KUKA KRL program: Glode_HanGao.src, Glode_HanGao.dat

--- Glode_HanGao.src ---
&ACCESS RVO1
&REL 298
&PARAM EDITMASK = *
&PARAM TEMPLATE = C:\KRC\Roboter\Template\vorgabe
&PARAM DISKPATH = KRC:\R1\Program\HK
DEF Glode_HanGao( )

;# DATE:2021-1-4



END

GLOBAL DEF HanGao_Surr_Calculate(Surr_Path:IN , Sink_Area:IN ,POS_Type:IN , Lin_Pos:OUt , Cir_Middle_POS:OUT , Cir_END_POS:OUT , Offset_info:OUT  ,Offset_cir_info:out , Offset_No:IN , Work_Area:IN, Sink_Type:IN)
;------------DECL_VALUE--------------
DECL REAL Surr_Path
DECL Sink_Type_Enum  Sink_Type
DECL Area_Enum Sink_Area
DECL E6POS Lin_Pos
DECL E6POS Cir_Middle_POS
DECL E6POS Cir_END_POS
DECL Pos_Type_Enum Pos_Type
DECL Offset_POS Offset_info , Offset_cir_info
DECL Surround_Welding_Type Sink_Welding_Size
DECL INT OFFSET_NO,Work_Area

;------------DECL_VALUE--------------





Lin_Pos={X 0,Y 0, Z 0,A 0,B 0,C 0}

Cir_Middle_POS={X 0,Y 0, Z 0,A 0,B 0,C 0}

Cir_END_POS={X 0,Y 0, Z 0,A 0,B 0,C 0}


switch Work_Area

CASE 1
Sink_Welding_Size=N1_Sink_Data

CASE 2
Sink_Welding_Size=N2_Sink_Data

ENDSWITCH



SWITCH Sink_Area

CASE #L0





 UL_Equation(N315_OFFSET_POS,N45_OFFSET_POS,(Surr_Path*0.01),Sink_Welding_Size.Sink_Size_R,Lin_Pos)



 ;Lin_Pos.X=Sink_Welding_Size.Sink_Size_Width+Sink_Welding_Size.Sink_Size_Down_Distance
 ;Lin_Pos.Y=(Sink_Welding_Size.Sink_Size_Long-Sink_Welding_Size.Sink_Size_R*2)* (1-(Surr_Path*0.01))+Sink_Welding_Size.Sink_Size_Left_Distance+Sink_Welding_Size.Sink_Size_R
 Lin_Pos.Z=-(Sink_Welding_Size.Sink_Size_Panel_Thick)

 Lin_Pos.A=0
 Lin_Pos.B=L0_Welding_Craft[Work_Area,OFFSET_NO].Welding_Angle
 Lin_Pos.C=0


L0_Welding_Craft[Work_Area,OFFSET_NO].Welding_Pos.X=Lin_Pos.X
L0_Welding_Craft[Work_Area,OFFSET_NO].Welding_Pos.Y=Lin_Pos.Y
L0_Welding_Craft[Work_Area,OFFSET_NO].Welding_Pos.Z=Lin_Pos.Z
L0_Welding_Craft[Work_Area,OFFSET_NO].Welding_Pos.A=Lin_Pos.A
L0_Welding_Craft[Work_Area,OFFSET_NO].Welding_Pos.B=Lin_Pos.B
L0_Welding_Craft[Work_Area,OFFSET_NO].Welding_Pos.C=Lin_Pos.C
CASE #C45


SWITCH Pos_Type

CASE #C_LIN_POS


UL_Equation(N315_OFFSET_POS,N45_OFFSET_POS,1,Sink_Welding_Size.Sink_Size_R,Lin_Pos)

;Lin_Pos.X=Sink_Welding_Size.Sink_Size_Width+Sink_Welding_Size.Sink_Size_Down_Distance
;Lin_Pos.Y=Sink_Welding_Size.Sink_Size_Left_Distance+Sink_Welding_Size.Sink_Size_R
Lin_Pos.Z=-(Sink_Welding_Size.Sink_Size_Panel_Thick)

Lin_Pos.A=0
Lin_Pos.B=C45_Welding_Craft[Work_Area,1].Welding_Angle
Lin_Pos.C=0

C45_Welding_Craft[Work_Area,1].Welding_Pos.X=Lin_Pos.X
C45_Welding_Craft[Work_Area,1].Welding_Pos.Y=Lin_Pos.Y
C45_Welding_Craft[Work_Area,1].Welding_Pos.Z=Lin_Pos.Z
C45_Welding_Craft[Work_Area,1].Welding_Pos.A=Lin_Pos.A
C45_Welding_Craft[Work_Area,1].Welding_Pos.B=Lin_Pos.B
C45_Welding_Craft[Work_Area,1].Welding_Pos.C=Lin_Pos.C

CASE #C_CIR_POS


 Cir_Middle_POS.X=N45_CIR_POS.x
 Cir_Middle_POS.Y=N45_CIR_POS.Y

 ;Cir_Middle_POS.x=Sink_Welding_Size.Sink_Size_Down_Distance+Sink_Welding_Size.Sink_Size_Width-Sink_Welding_Size.Sink_Size_R+(COS(45)*Sink_Welding_Size.Sink_Size_R)
 ;Cir_Middle_POS.Y=Sink_Welding_Size.Sink_Size_Left_Distance+((1-COS(45))*Sink_Welding_Size.Sink_Size_R)
 Cir_Middle_POS.Z=-(Sink_Welding_Size.Sink_Size_Panel_Thick)


 UL_Equation(N45_OFFSET_POS,N135_OFFSET_POS,0,Sink_Welding_Size.Sink_Size_R,Cir_END_POS)

 ;Cir_END_POS.X=Sink_Welding_Size.Sink_Size_Down_Distance+Sink_Welding_Size.Sink_Size_Width-Sink_Welding_Size.Sink_Size_R
 ;Cir_END_POS.Y=Sink_Welding_Size.Sink_Size_Left_Distance
 Cir_END_POS.Z=-(Sink_Welding_Size.Sink_Size_Panel_Thick)


 Cir_END_POS.A=0
 Cir_END_POS.B=0
 Cir_END_POS.C=C45_Welding_Craft[Work_Area,3].Welding_Angle



C45_Welding_Craft[Work_Area,2].Welding_Pos.X=Cir_Middle_POS.X
C45_Welding_Craft[Work_Area,2].Welding_Pos.Y=Cir_Middle_POS.Y
C45_Welding_Craft[Work_Area,2].Welding_Pos.Z=Cir_Middle_POS.Z
C45_Welding_Craft[Work_Area,2].Welding_Pos.A=Cir_Middle_POS.A
C45_Welding_Craft[Work_Area,2].Welding_Pos.B=Cir_Middle_POS.B
C45_Welding_Craft[Work_Area,2].Welding_Pos.C=Cir_Middle_POS.C

C45_Welding_Craft[Work_Area,3].Welding_Pos.X=Cir_END_POS.X
C45_Welding_Craft[Work_Area,3].Welding_Pos.Y=Cir_END_POS.Y
C45_Welding_Craft[Work_Area,3].Welding_Pos.Z=Cir_END_POS.Z
C45_Welding_Craft[Work_Area,3].Welding_Pos.A=Cir_END_POS.A
C45_Welding_Craft[Work_Area,3].Welding_Pos.B=Cir_END_POS.B
C45_Welding_Craft[Work_Area,3].Welding_Pos.C=Cir_END_POS.C

ENDSWITCH


CASE #L90


UL_Equation(N45_OFFSET_POS,N135_OFFSET_POS,(Surr_Path*0.01),Sink_Welding_Size.Sink_Size_R, Lin_Pos)

 ;Lin_Pos.X=(Sink_Welding_Size.Sink_Size_Width-Sink_Welding_Size.Sink_Size_R*2)* (1-(Surr_Path*0.01))+Sink_Welding_Size.Sink_Size_Down_Distance+Sink_Welding_Size.Sink_Size_R
 ;Lin_Pos.Y=Sink_Welding_Size.Sink_Size_Left_Distance
 Lin_Pos.Z=-(Sink_Welding_Size.Sink_Size_Panel_Thick)
 Lin_Pos.A=0
 Lin_Pos.B=0
 Lin_Pos.C=L90_Welding_Craft[Work_Area,OFFSET_NO].Welding_Angle

L90_Welding_Craft[Work_Area,OFFSET_NO].Welding_Pos.X=Lin_Pos.X
L90_Welding_Craft[Work_Area,OFFSET_NO].Welding_Pos.Y=Lin_Pos.Y
L90_Welding_Craft[Work_Area,OFFSET_NO].Welding_Pos.Z=Lin_Pos.Z
L90_Welding_Craft[Work_Area,OFFSET_NO].Welding_Pos.A=Lin_Pos.A
L90_Welding_Craft[Work_Area,OFFSET_NO].Welding_Pos.B=Lin_Pos.B
L90_Welding_Craft[Work_Area,OFFSET_NO].Welding_Pos.C=Lin_Pos.C

CASE #C135

SWITCH Pos_Type

CASE #C_LIN_POS

UL_Equation(N45_OFFSET_POS,N135_OFFSET_POS,1,Sink_Welding_Size.Sink_Size_R, Lin_Pos)

 ;Lin_Pos.X=Sink_Welding_Size.Sink_Size_Down_Distance+Sink_Welding_Size.Sink_Size_R
 ;Lin_Pos.Y=Sink_Welding_Size.Sink_Size_Left_Distance
 Lin_Pos.Z=-(Sink_Welding_Size.Sink_Size_Panel_Thick)
 Lin_Pos.A=0
 Lin_Pos.B=0
 Lin_Pos.C=C135_Welding_Craft[Work_Area,1].Welding_Angle

C135_Welding_Craft[Work_Area,1].Welding_Pos.X=Lin_Pos.X
C135_Welding_Craft[Work_Area,1].Welding_Pos.Y=Lin_Pos.Y
C135_Welding_Craft[Work_Area,1].Welding_Pos.Z=Lin_Pos.Z
C135_Welding_Craft[Work_Area,1].Welding_Pos.A=Lin_Pos.A
C135_Welding_Craft[Work_Area,1].Welding_Pos.B=Lin_Pos.B
C135_Welding_Craft[Work_Area,1].Welding_Pos.C=Lin_Pos.C

CASE #C_CIR_POS



 Cir_Middle_POS.X=N135_CIR_POS.x
 Cir_Middle_POS.Y=N135_CIR_POS.Y


 ;Cir_Middle_POS.x=Sink_Welding_Size.Sink_Size_Down_Distance+((1-COS(45))*Sink_Welding_Size.Sink_Size_R)
 ;Cir_Middle_POS.Y=Sink_Welding_Size.Sink_Size_Left_Distance+((1-COS(45))*Sink_Welding_Size.Sink_Size_R)
 Cir_Middle_POS.Z=-(Sink_Welding_Size.Sink_Size_Panel_Thick)



 UL_Equation(N135_OFFSET_POS,N225_OFFSET_POS,0,Sink_Welding_Size.Sink_Size_R,Cir_END_POS)

 ;Cir_END_POS.X=Sink_Welding_Size.Sink_Size_Down_Distance
 ;Cir_END_POS.Y=Sink_Welding_Size.Sink_Size_Left_Distance+Sink_Welding_Size.Sink_Size_R
 Cir_END_POS.Z=-(Sink_Welding_Size.Sink_Size_Panel_Thick)
 Cir_END_POS.A=0
 Cir_END_POS.B=C135_Welding_Craft[Work_Area,3].Welding_Angle
 Cir_END_POS.C=0

C135_Welding_Craft[Work_Area,2].Welding_Pos.X=Cir_Middle_POS.X
C135_Welding_Craft[Work_Area,2].Welding_Pos.Y=Cir_Middle_POS.Y
C135_Welding_Craft[Work_Area,2].Welding_Pos.Z=Cir_Middle_POS.Z
C135_Welding_Craft[Work_Area,2].Welding_Pos.A=Cir_Middle_POS.A
C135_Welding_Craft[Work_Area,2].Welding_Pos.B=Cir_Middle_POS.B
C135_Welding_Craft[Work_Area,2].Welding_Pos.C=Cir_Middle_POS.C

C135_Welding_Craft[Work_Area,3].Welding_Pos.X=Cir_END_POS.X
C135_Welding_Craft[Work_Area,3].Welding_Pos.Y=Cir_END_POS.Y
C135_Welding_Craft[Work_Area,3].Welding_Pos.Z=Cir_END_POS.Z
C135_Welding_Craft[Work_Area,3].Welding_Pos.A=Cir_END_POS.A
C135_Welding_Craft[Work_Area,3].Welding_Pos.B=Cir_END_POS.B
C135_Welding_Craft[Work_Area,3].Welding_Pos.C=Cir_END_POS.C

ENDSWITCH


CASE #L180

UL_Equation(N135_OFFSET_POS,N225_OFFSET_POS,(Surr_Path*0.01),Sink_Welding_Size.Sink_Size_R, Lin_Pos)

 ;Lin_Pos.X=Sink_Welding_Size.Sink_Size_Down_Distance
 ;Lin_Pos.Y=(Sink_Welding_Size.Sink_Size_Long-Sink_Welding_Size.Sink_Size_R*2)* (Surr_Path*0.01)+Sink_Welding_Size.Sink_Size_Left_Distance+Sink_Welding_Size.Sink_Size_R
 Lin_Pos.Z=-(Sink_Welding_Size.Sink_Size_Panel_Thick)
 Lin_Pos.A=0
 Lin_Pos.B=L180_Welding_Craft[Work_Area,OFFSET_NO].Welding_Angle
 Lin_Pos.C=0

L180_Welding_Craft[Work_Area,OFFSET_NO].Welding_Pos.X=Lin_Pos.X
L180_Welding_Craft[Work_Area,OFFSET_NO].Welding_Pos.Y=Lin_Pos.Y
L180_Welding_Craft[Work_Area,OFFSET_NO].Welding_Pos.Z=Lin_Pos.Z
L180_Welding_Craft[Work_Area,OFFSET_NO].Welding_Pos.A=Lin_Pos.A
L180_Welding_Craft[Work_Area,OFFSET_NO].Welding_Pos.B=Lin_Pos.B
L180_Welding_Craft[Work_Area,OFFSET_NO].Welding_Pos.C=Lin_Pos.C

CASE #C225

SWITCH Pos_Type

CASE #C_LIN_POS


 UL_Equation(N135_OFFSET_POS,N225_OFFSET_POS,1,Sink_Welding_Size.Sink_Size_R, Lin_Pos)

 ;Lin_Pos.X=Sink_Welding_Size.Sink_Size_Down_Distance
 ;Lin_Pos.Y=Sink_Welding_Size.Sink_Size_Left_Distance+Sink_Welding_Size.Sink_Size_Long-Sink_Welding_Size.Sink_Size_R
 Lin_Pos.Z=-(Sink_Welding_Size.Sink_Size_Panel_Thick)
 Lin_Pos.A=0
 Lin_Pos.B=C225_Welding_Craft[Work_Area,1].Welding_Angle
 Lin_Pos.C=0

C225_Welding_Craft[Work_Area,1].Welding_Pos.X=Lin_Pos.X
C225_Welding_Craft[Work_Area,1].Welding_Pos.Y=Lin_Pos.Y
C225_Welding_Craft[Work_Area,1].Welding_Pos.Z=Lin_Pos.Z
C225_Welding_Craft[Work_Area,1].Welding_Pos.A=Lin_Pos.A
C225_Welding_Craft[Work_Area,1].Welding_Pos.B=Lin_Pos.B
C225_Welding_Craft[Work_Area,1].Welding_Pos.C=Lin_Pos.C

CASE #C_CIR_POS


 Cir_Middle_POS.X=N225_CIR_POS.x
 Cir_Middle_POS.Y=N225_CIR_POS.Y




 ;Cir_Middle_POS.x=Sink_Welding_Size.Sink_Size_Down_Distance+((1-COS(45))*Sink_Welding_Size.Sink_Size_R)
 ;Cir_Middle_POS.Y=Sink_Welding_Size.Sink_Size_Left_Distance+Sink_Welding_Size.Sink_Size_Long-Sink_Welding_Size.Sink_Size_R+( COS(45)*Sink_Welding_Size.Sink_Size_R )
 Cir_Middle_POS.Z=-(Sink_Welding_Size.Sink_Size_Panel_Thick)

  UL_Equation(N225_OFFSET_POS,N315_OFFSET_POS,0,Sink_Welding_Size.Sink_Size_R,Cir_END_POS)

 ;Cir_END_POS.X=Sink_Welding_Size.Sink_Size_Down_Distance+Sink_Welding_Size.Sink_Size_R
; Cir_END_POS.Y=Sink_Welding_Size.Sink_Size_Left_Distance+Sink_Welding_Size.Sink_Size_Long
 Cir_END_POS.Z=-(Sink_Welding_Size.Sink_Size_Panel_Thick)
 Cir_END_POS.A=0
 Cir_END_POS.B=0
 Cir_END_POS.C=C225_Welding_Craft[Work_Area,3].Welding_Angle

C225_Welding_Craft[Work_Area,2].Welding_Pos.X=Cir_Middle_POS.X
C225_Welding_Craft[Work_Area,2].Welding_Pos.Y=Cir_Middle_POS.Y
C225_Welding_Craft[Work_Area,2].Welding_Pos.Z=Cir_Middle_POS.Z
C225_Welding_Craft[Work_Area,2].Welding_Pos.A=Cir_Middle_POS.A
C225_Welding_Craft[Work_Area,2].Welding_Pos.B=Cir_Middle_POS.B
C225_Welding_Craft[Work_Area,2].Welding_Pos.C=Cir_Middle_POS.C

C225_Welding_Craft[Work_Area,3].Welding_Pos.X=Cir_END_POS.X
C225_Welding_Craft[Work_Area,3].Welding_Pos.Y=Cir_END_POS.Y
C225_Welding_Craft[Work_Area,3].Welding_Pos.Z=Cir_END_POS.Z
C225_Welding_Craft[Work_Area,3].Welding_Pos.A=Cir_END_POS.A
C225_Welding_Craft[Work_Area,3].Welding_Pos.B=Cir_END_POS.B
C225_Welding_Craft[Work_Area,3].Welding_Pos.C=Cir_END_POS.C

ENDSWITCH


CASE #L270



UL_Equation(N225_OFFSET_POS,N315_OFFSET_POS,(Surr_Path*0.01),Sink_Welding_Size.Sink_Size_R, Lin_Pos)




; Lin_Pos.X=(Sink_Welding_Size.Sink_Size_Width-Sink_Welding_Size.Sink_Size_R*2)* (Surr_Path*0.01)+Sink_Welding_Size.Sink_Size_Down_Distance+Sink_Welding_Size.Sink_Size_R
 ;Lin_Pos.Y=Sink_Welding_Size.Sink_Size_Left_Distance+Sink_Welding_Size.Sink_Size_Long
 Lin_Pos.Z=-(Sink_Welding_Size.Sink_Size_Panel_Thick)
 Lin_Pos.A=0
 Lin_Pos.B=0
 Lin_Pos.C=L270_Welding_Craft[Work_Area,OFFSET_NO].Welding_Angle

L270_Welding_Craft[Work_Area,OFFSET_NO].Welding_Pos.X=Lin_Pos.X
L270_Welding_Craft[Work_Area,OFFSET_NO].Welding_Pos.Y=Lin_Pos.Y
L270_Welding_Craft[Work_Area,OFFSET_NO].Welding_Pos.Z=Lin_Pos.Z
L270_Welding_Craft[Work_Area,OFFSET_NO].Welding_Pos.A=Lin_Pos.A
L270_Welding_Craft[Work_Area,OFFSET_NO].Welding_Pos.B=Lin_Pos.B
L270_Welding_Craft[Work_Area,OFFSET_NO].Welding_Pos.C=Lin_Pos.C

CASE #C315

SWITCH Pos_Type

CASE #C_LIN_POS



 UL_Equation(N225_OFFSET_POS,N315_OFFSET_POS,1,Sink_Welding_Size.Sink_Size_R, Lin_Pos)




 ;Lin_Pos.X=Sink_Welding_Size.Sink_Size_Down_Distance+Sink_Welding_Size.Sink_Size_Width-Sink_Welding_Size.Sink_Size_R
 ;Lin_Pos.Y=Sink_Welding_Size.Sink_Size_Long+Sink_Welding_Size.Sink_Size_Left_Distance
 Lin_Pos.Z=-(Sink_Welding_Size.Sink_Size_Panel_Thick)
 Lin_Pos.A=0
 Lin_Pos.B=0
 Lin_Pos.C=C315_Welding_Craft[Work_Area,1].Welding_Angle

 C315_Welding_Craft[Work_Area,1].Welding_Pos.X=Lin_Pos.X
 C315_Welding_Craft[Work_Area,1].Welding_Pos.Y=Lin_Pos.Y
 C315_Welding_Craft[Work_Area,1].Welding_Pos.Z=Lin_Pos.Z
 C315_Welding_Craft[Work_Area,1].Welding_Pos.A=Lin_Pos.A
 C315_Welding_Craft[Work_Area,1].Welding_Pos.B=Lin_Pos.B
 C315_Welding_Craft[Work_Area,1].Welding_Pos.C=Lin_Pos.C

CASE #C_CIR_POS


 Cir_Middle_POS.X=N315_CIR_POS.x
 Cir_Middle_POS.Y=N315_CIR_POS.Y


 ;Cir_Middle_POS.x=Sink_Welding_Size.Sink_Size_Down_Distance+Sink_Welding_Size.Sink_Size_Width-Sink_Welding_Size.Sink_Size_R+(COS(45)*Sink_Welding_Size.Sink_Size_R)
 ;Cir_Middle_POS.Y=Sink_Welding_Size.Sink_Size_Long+Sink_Welding_Size.Sink_Size_Left_Distance-Sink_Welding_Size.Sink_Size_R+(COS(45)*Sink_Welding_Size.Sink_Size_R)
 Cir_Middle_POS.Z=-(Sink_Welding_Size.Sink_Size_Panel_Thick)

   UL_Equation(N315_OFFSET_POS,N45_OFFSET_POS,0,Sink_Welding_Size.Sink_Size_R,Cir_END_POS)

 ;Cir_END_POS.X=Sink_Welding_Size.Sink_Size_Down_Distance+Sink_Welding_Size.Sink_Size_Width
 ;Cir_END_POS.Y=Sink_Welding_Size.Sink_Size_Left_Distance+Sink_Welding_Size.Sink_Size_Long-Sink_Welding_Size.Sink_Size_R
 Cir_END_POS.Z=-(Sink_Welding_Size.Sink_Size_Panel_Thick)
 Cir_END_POS.A=0
 Cir_END_POS.B=C315_Welding_Craft[Work_Area,3].Welding_Angle
 Cir_END_POS.C=0

C315_Welding_Craft[Work_Area,2].Welding_Pos.X=Cir_Middle_POS.X
C315_Welding_Craft[Work_Area,2].Welding_Pos.Y=Cir_Middle_POS.Y
C315_Welding_Craft[Work_Area,2].Welding_Pos.Z=Cir_Middle_POS.Z
C315_Welding_Craft[Work_Area,2].Welding_Pos.A=Cir_Middle_POS.A
C315_Welding_Craft[Work_Area,2].Welding_Pos.B=Cir_Middle_POS.B
C315_Welding_Craft[Work_Area,2].Welding_Pos.C=Cir_Middle_POS.C

C315_Welding_Craft[Work_Area,3].Welding_Pos.X=Cir_END_POS.X
C315_Welding_Craft[Work_Area,3].Welding_Pos.Y=Cir_END_POS.Y
C315_Welding_Craft[Work_Area,3].Welding_Pos.Z=Cir_END_POS.Z
C315_Welding_Craft[Work_Area,3].Welding_Pos.A=Cir_END_POS.A
C315_Welding_Craft[Work_Area,3].Welding_Pos.B=Cir_END_POS.B
C315_Welding_Craft[Work_Area,3].Welding_Pos.C=Cir_END_POS.C

ENDSWITCH





CASE #N45
;




SWITCH  Offset_No

CASE 1

SWITCH Sink_Welding_Size.Sink_Type
CASE #UpDown_One

Lin_Pos.X=D45_Start_POS.X
Lin_Pos.Y=D45_Start_POS.X

;Lin_Pos.X=Sink_Welding_Size.Sink_Size_Down_Distance*2+Sink_Welding_Size.Sink_Size_Width
;Lin_Pos.Y=Sink_Welding_Size.Sink_Size_Short_TwoPos
Lin_Pos.Z=-150.000
Lin_Pos.A=0
Lin_Pos.B=0
Lin_Pos.C=0
case #LeftRight_One

Lin_Pos.X=D45_Start_POS.X
Lin_Pos.Y=D45_Start_POS.Y

;Lin_Pos.X=Sink_Welding_Size.Sink_Size_Short_OnePos+Sink_Welding_Size.Sink_Size_Short_TwoPos
;Lin_Pos.Y=0
Lin_Pos.Z=-150.000
Lin_Pos.A=0
Lin_Pos.B=0
Lin_Pos.C=0
ENDSWITCH

N45_Short_Craft[Work_Area,1].Welding_Pos.X=Lin_Pos.X
N45_Short_Craft[Work_Area,1].Welding_Pos.Y=Lin_Pos.Y
N45_Short_Craft[Work_Area,1].Welding_Pos.Z=Lin_Pos.Z
N45_Short_Craft[Work_Area,1].Welding_Pos.A=Lin_Pos.A
N45_Short_Craft[Work_Area,1].Welding_Pos.B=Lin_Pos.B
N45_Short_Craft[Work_Area,1].Welding_Pos.C=Lin_Pos.C

CASE 2
SWITCH Sink_Welding_Size.Sink_Type
CASE #UpDown_One

Lin_Pos.X=D45_Start_POS.X
Lin_Pos.Y=D45_Start_POS.Y

;Lin_Pos.X=Sink_Welding_Size.Sink_Size_Down_Distance*2+Sink_Welding_Size.Sink_Size_Width
;Lin_Pos.Y=Sink_Welding_Size.Sink_Size_Short_TwoPos
Lin_Pos.Z=0
Lin_Pos.A=0
Lin_Pos.B=0
Lin_Pos.C=0
case #LeftRight_One

Lin_Pos.X=D45_Start_POS.X
Lin_Pos.Y=D45_Start_POS.Y

; Lin_Pos.X=Sink_Welding_Size.Sink_Size_Short_OnePos+Sink_Welding_Size.Sink_Size_Short_TwoPos
; Lin_Pos.Y=0
Lin_Pos.Z=0
Lin_Pos.A=0
Lin_Pos.B=0
Lin_Pos.C=0
ENDSWITCH


N45_Short_Craft[Work_Area,2].Welding_Pos.X=Lin_Pos.X
N45_Short_Craft[Work_Area,2].Welding_Pos.Y=Lin_Pos.Y
N45_Short_Craft[Work_Area,2].Welding_Pos.Z=Lin_Pos.Z
N45_Short_Craft[Work_Area,2].Welding_Pos.A=Lin_Pos.A
N45_Short_Craft[Work_Area,2].Welding_Pos.B=Lin_Pos.B
N45_Short_Craft[Work_Area,2].Welding_Pos.C=Lin_Pos.C

CASE 3
SWITCH Sink_Welding_Size.Sink_Type
CASE #UpDown_One

Lin_Pos.X=D45_End_POS.X
Lin_Pos.Y=D45_End_POS.Y

;Lin_Pos.X=Sink_Welding_Size.Sink_Size_Down_Distance*2+Sink_Welding_Size.Sink_Size_Width
;Lin_Pos.Y=Sink_Welding_Size.Sink_Size_Short_TwoPos-Sink_Welding_Size.Sink_Size_Short_Side
Lin_Pos.Z=0.000
Lin_Pos.A=0
Lin_Pos.B=0
Lin_Pos.C=0
case #LeftRight_One

Lin_Pos.X=D45_End_POS.X
Lin_Pos.Y=D45_End_POS.Y

;Lin_Pos.X=Sink_Welding_Size.Sink_Size_Short_OnePos+Sink_Welding_Size.Sink_Size_Short_TwoPos
;Lin_Pos.Y=Sink_Welding_Size.Sink_Size_Short_Side
Lin_Pos.Z=0.000
Lin_Pos.A=0
Lin_Pos.B=0
Lin_Pos.C=0
ENDSWITCH


N45_Short_Craft[Work_Area,3].Welding_Pos.X=Lin_Pos.X
N45_Short_Craft[Work_Area,3].Welding_Pos.Y=Lin_Pos.Y
N45_Short_Craft[Work_Area,3].Welding_Pos.Z=Lin_Pos.Z
N45_Short_Craft[Work_Area,3].Welding_Pos.A=Lin_Pos.A
N45_Short_Craft[Work_Area,3].Welding_Pos.B=Lin_Pos.B
N45_Short_Craft[Work_Area,3].Welding_Pos.C=Lin_Pos.C

CASE 4
SWITCH Sink_Welding_Size.Sink_Type
CASE #UpDown_One

UL_Equation(D45_Start_POS,D45_End_POS,(Surr_Path*0.01),Sink_Welding_Size.Sink_Size_R,Lin_Pos)

;Lin_Pos.X=Sink_Welding_Size.Sink_Size_Down_Distance+Sink_Welding_Size.Sink_Size_Width+Sink_Welding_Size.Sink_Size_Short_Side*(Surr_Path/100)
;Lin_Pos.Y=Sink_Welding_Size.Sink_Size_Short_TwoPos-Sink_Welding_Size.Sink_Size_Short_Side
Lin_Pos.Z=-150
Lin_Pos.A=0
Lin_Pos.B=0
Lin_Pos.C=0
case #LeftRight_One

UL_Equation(D45_Start_POS,D45_End_POS,(Surr_Path*0.01),Sink_Welding_Size.Sink_Size_R,Lin_Pos)

;Lin_Pos.X=Sink_Welding_Size.Sink_Size_Short_OnePos+Sink_Welding_Size.Sink_Size_Short_TwoPos
;Lin_Pos.Y=Sink_Welding_Size.Sink_Size_Short_Side-Sink_Welding_Size.Sink_Size_Short_Side*(Surr_Path/100)
Lin_Pos.Z=-150
Lin_Pos.A=0
Lin_Pos.B=0
Lin_Pos.C=0
ENDSWITCH


N45_Short_Craft[Work_Area,4].Welding_Pos.X=Lin_Pos.X
N45_Short_Craft[Work_Area,4].Welding_Pos.Y=Lin_Pos.Y
N45_Short_Craft[Work_Area,4].Welding_Pos.Z=Lin_Pos.Z
N45_Short_Craft[Work_Area,4].Welding_Pos.A=Lin_Pos.A
N45_Short_Craft[Work_Area,4].Welding_Pos.B=Lin_Pos.B
N45_Short_Craft[Work_Area,4].Welding_Pos.C=Lin_Pos.C
ENDSWITCH






CASE #N135
;
SWITCH  Offset_No

CASE 1
SWITCH Sink_Welding_Size.Sink_Type
CASE #UpDown_One

Lin_Pos.X=D135_Start_POS.X
Lin_Pos.Y=D135_Start_POS.Y

;Lin_Pos.X=0
;Lin_Pos.Y=Sink_Welding_Size.Sink_Size_Short_OnePos
Lin_Pos.Z=-150.000
Lin_Pos.A=0
Lin_Pos.B=0
Lin_Pos.C=0
case #LeftRight_One

Lin_Pos.X=D135_Start_POS.X
Lin_Pos.Y=D135_Start_POS.Y

;Lin_Pos.X=Sink_Welding_Size.Sink_Size_Short_OnePos
;Lin_Pos.Y=0
Lin_Pos.Z=-150.000
Lin_Pos.A=0
Lin_Pos.B=0
Lin_Pos.C=0
ENDSWITCH


N135_Short_Craft[Work_Area,1].Welding_Pos.X=Lin_Pos.X
N135_Short_Craft[Work_Area,1].Welding_Pos.Y=Lin_Pos.Y
N135_Short_Craft[Work_Area,1].Welding_Pos.Z=Lin_Pos.Z
N135_Short_Craft[Work_Area,1].Welding_Pos.A=Lin_Pos.A
N135_Short_Craft[Work_Area,1].Welding_Pos.B=Lin_Pos.B
N135_Short_Craft[Work_Area,1].Welding_Pos.C=Lin_Pos.C

CASE 2
SWITCH Sink_Welding_Size.Sink_Type
CASE #UpDown_One

Lin_Pos.X=D135_Start_POS.X
Lin_Pos.Y=D135_Start_POS.Y

;Lin_Pos.X=0
;Lin_Pos.Y=Sink_Welding_Size.Sink_Size_Short_OnePos
Lin_Pos.Z=0
Lin_Pos.A=0
Lin_Pos.B=0
Lin_Pos.C=0
case #LeftRight_One

Lin_Pos.X=D135_Start_POS.X
Lin_Pos.Y=D135_Start_POS.Y

;Lin_Pos.X=Sink_Welding_Size.Sink_Size_Short_OnePos
;Lin_Pos.Y=0
Lin_Pos.Z=0
Lin_Pos.A=0
Lin_Pos.B=0
Lin_Pos.C=0
ENDSWITCH


N135_Short_Craft[Work_Area,2].Welding_Pos.X=Lin_Pos.X
N135_Short_Craft[Work_Area,2].Welding_Pos.Y=Lin_Pos.Y
N135_Short_Craft[Work_Area,2].Welding_Pos.Z=Lin_Pos.Z
N135_Short_Craft[Work_Area,2].Welding_Pos.A=Lin_Pos.A
N135_Short_Craft[Work_Area,2].Welding_Pos.B=Lin_Pos.B
N135_Short_Craft[Work_Area,2].Welding_Pos.C=Lin_Pos.C
CASE 3
SWITCH Sink_Welding_Size.Sink_Type
CASE #UpDown_One

Lin_Pos.X=D135_End_POS.X
Lin_Pos.Y=D135_End_POS.Y

;Lin_Pos.X=Sink_Welding_Size.Sink_Size_Short_Side
;Lin_Pos.Y=Sink_Welding_Size.Sink_Size_Short_OnePos
Lin_Pos.Z=0.000
Lin_Pos.A=0
Lin_Pos.B=0
Lin_Pos.C=0
case #LeftRight_One

Lin_Pos.X=D135_End_POS.X
Lin_Pos.Y=D135_End_POS.Y

;Lin_Pos.X=Sink_Welding_Size.Sink_Size_Short_OnePos
;Lin_Pos.Y=Sink_Welding_Size.Sink_Size_Short_Side
Lin_Pos.Z=0.000
Lin_Pos.A=0
Lin_Pos.B=0
Lin_Pos.C=0
ENDSWITCH


N135_Short_Craft[Work_Area,3].Welding_Pos.X=Lin_Pos.X
N135_Short_Craft[Work_Area,3].Welding_Pos.Y=Lin_Pos.Y
N135_Short_Craft[Work_Area,3].Welding_Pos.Z=Lin_Pos.Z
N135_Short_Craft[Work_Area,3].Welding_Pos.A=Lin_Pos.A
N135_Short_Craft[Work_Area,3].Welding_Pos.B=Lin_Pos.B
N135_Short_Craft[Work_Area,3].Welding_Pos.C=Lin_Pos.C
CASE 4
SWITCH Sink_Welding_Size.Sink_Type
CASE #UpDown_One


UL_Equation(D135_Start_POS,D135_End_POS,(Surr_Path*0.01),Sink_Welding_Size.Sink_Size_R,Lin_Pos)

;Lin_Pos.X=Sink_Welding_Size.Sink_Size_Short_Side-Sink_Welding_Size.Sink_Size_Short_Side*(Surr_Path/100)
;Lin_Pos.Y=Sink_Welding_Size.Sink_Size_Short_OnePos
Lin_Pos.Z=-150.000
Lin_Pos.A=0
Lin_Pos.B=0
Lin_Pos.C=0
case #LeftRight_One

UL_Equation(D135_Start_POS,D135_End_POS,(Surr_Path*0.01),Sink_Welding_Size.Sink_Size_R,Lin_Pos)

;Lin_Pos.X=Sink_Welding_Size.Sink_Size_Short_OnePos
;Lin_Pos.Y=Sink_Welding_Size.Sink_Size_Short_Side-Sink_Welding_Size.Sink_Size_Short_Side*(Surr_Path/100)
Lin_Pos.Z=-150.000
Lin_Pos.A=0
Lin_Pos.B=0
Lin_Pos.C=0
ENDSWITCH


N135_Short_Craft[Work_Area,4].Welding_Pos.X=Lin_Pos.X
N135_Short_Craft[Work_Area,4].Welding_Pos.Y=Lin_Pos.Y
N135_Short_Craft[Work_Area,4].Welding_Pos.Z=Lin_Pos.Z
N135_Short_Craft[Work_Area,4].Welding_Pos.A=Lin_Pos.A
N135_Short_Craft[Work_Area,4].Welding_Pos.B=Lin_Pos.B
N135_Short_Craft[Work_Area,4].Welding_Pos.C=Lin_Pos.C

ENDSWITCH





CASE #N225
;
SWITCH  Offset_No

CASE 1
SWITCH Sink_Welding_Size.Sink_Type
CASE #UpDown_One

Lin_Pos.X=D225_Start_POS.X
Lin_Pos.Y=D225_Start_POS.Y

;Lin_Pos.X=0
;Lin_Pos.Y=Sink_Welding_Size.Sink_Size_Short_OnePos+Sink_Welding_Size.Sink_Size_Short_TwoPos
Lin_Pos.Z=-150.000
Lin_Pos.A=0
Lin_Pos.B=0
Lin_Pos.C=0
case #LeftRight_One

Lin_Pos.X=D225_Start_POS.X
Lin_Pos.Y=D225_Start_POS.Y

;Lin_Pos.X=Sink_Welding_Size.Sink_Size_Short_OnePos
;Lin_Pos.Y=Sink_Welding_Size.Sink_Size_Long+Sink_Welding_Size.Sink_Size_Left_Distance*2
Lin_Pos.Z=-150.000
Lin_Pos.A=0
Lin_Pos.B=0
Lin_Pos.C=0
ENDSWITCH


N225_Short_Craft[Work_Area,1].Welding_Pos.X=Lin_Pos.X
N225_Short_Craft[Work_Area,1].Welding_Pos.Y=Lin_Pos.Y
N225_Short_Craft[Work_Area,1].Welding_Pos.Z=Lin_Pos.Z
N225_Short_Craft[Work_Area,1].Welding_Pos.A=Lin_Pos.A
N225_Short_Craft[Work_Area,1].Welding_Pos.B=Lin_Pos.B
N225_Short_Craft[Work_Area,1].Welding_Pos.C=Lin_Pos.C

CASE 2
SWITCH Sink_Welding_Size.Sink_Type
CASE #UpDown_One

Lin_Pos.X=D225_Start_POS.X
Lin_Pos.Y=D225_Start_POS.Y

;Lin_Pos.X=0
;Lin_Pos.Y=Sink_Welding_Size.Sink_Size_Short_OnePos+Sink_Welding_Size.Sink_Size_Short_TwoPos
Lin_Pos.Z=0
Lin_Pos.A=0
Lin_Pos.B=0
Lin_Pos.C=0
case #LeftRight_One

Lin_Pos.X=D225_Start_POS.X
Lin_Pos.Y=D225_Start_POS.Y

;Lin_Pos.X=Sink_Welding_Size.Sink_Size_Short_OnePos
;Lin_Pos.Y=Sink_Welding_Size.Sink_Size_Long+Sink_Welding_Size.Sink_Size_Left_Distance*2
Lin_Pos.Z=0
Lin_Pos.A=0
Lin_Pos.B=0
Lin_Pos.C=0
ENDSWITCH


N225_Short_Craft[Work_Area,2].Welding_Pos.X=Lin_Pos.X
N225_Short_Craft[Work_Area,2].Welding_Pos.Y=Lin_Pos.Y
N225_Short_Craft[Work_Area,2].Welding_Pos.Z=Lin_Pos.Z
N225_Short_Craft[Work_Area,2].Welding_Pos.A=Lin_Pos.A
N225_Short_Craft[Work_Area,2].Welding_Pos.B=Lin_Pos.B
N225_Short_Craft[Work_Area,2].Welding_Pos.C=Lin_Pos.C

CASE 3
SWITCH Sink_Welding_Size.Sink_Type
CASE #UpDown_One


Lin_Pos.X=D225_End_POS.X
Lin_Pos.Y=D225_End_POS.Y

;Lin_Pos.X=Sink_Welding_Size.Sink_Size_Short_Side
;Lin_Pos.Y=Sink_Welding_Size.Sink_Size_Short_OnePos+Sink_Welding_Size.Sink_Size_Short_TwoPos
Lin_Pos.Z=0
Lin_Pos.A=0
Lin_Pos.B=0
Lin_Pos.C=0
case #LeftRight_One

Lin_Pos.X=D225_End_POS.X
Lin_Pos.Y=D225_End_POS.Y

;Lin_Pos.X=Sink_Welding_Size.Sink_Size_Short_OnePos
;Lin_Pos.Y=Sink_Welding_Size.Sink_Size_Long+Sink_Welding_Size.Sink_Size_Left_Distance*2-Sink_Welding_Size.Sink_Size_Short_Side
Lin_Pos.Z=0
Lin_Pos.A=0
Lin_Pos.B=0
Lin_Pos.C=0
ENDSWITCH


N225_Short_Craft[Work_Area,3].Welding_Pos.X=Lin_Pos.X
N225_Short_Craft[Work_Area,3].Welding_Pos.Y=Lin_Pos.Y
N225_Short_Craft[Work_Area,3].Welding_Pos.Z=Lin_Pos.Z
N225_Short_Craft[Work_Area,3].Welding_Pos.A=Lin_Pos.A
N225_Short_Craft[Work_Area,3].Welding_Pos.B=Lin_Pos.B
N225_Short_Craft[Work_Area,3].Welding_Pos.C=Lin_Pos.C

CASE 4
SWITCH Sink_Welding_Size.Sink_Type
CASE #UpDown_One

UL_Equation(D225_Start_POS,D225_End_POS,(Surr_Path*0.01),Sink_Welding_Size.Sink_Size_R,Lin_Pos)

;Lin_Pos.X=Sink_Welding_Size.Sink_Size_Short_Side-Sink_Welding_Size.Sink_Size_Short_Side*(Surr_Path/100)
;Lin_Pos.Y=Sink_Welding_Size.Sink_Size_Short_OnePos+Sink_Welding_Size.Sink_Size_Short_TwoPos
Lin_Pos.Z=-150.000
Lin_Pos.A=0
Lin_Pos.B=0
Lin_Pos.C=0
case #LeftRight_One

UL_Equation(D225_Start_POS,D225_End_POS,(Surr_Path*0.01),Sink_Welding_Size.Sink_Size_R,Lin_Pos)

;Lin_Pos.X=Sink_Welding_Size.Sink_Size_Short_OnePos
;Lin_Pos.Y=Sink_Welding_Size.Sink_Size_Long+Sink_Welding_Size.Sink_Size_Left_Distance+Sink_Welding_Size.Sink_Size_Short_Side*(Surr_Path/100)
Lin_Pos.Z=-150.000
Lin_Pos.A=0
Lin_Pos.B=0
Lin_Pos.C=0
ENDSWITCH


N225_Short_Craft[Work_Area,4].Welding_Pos.X=Lin_Pos.X
N225_Short_Craft[Work_Area,4].Welding_Pos.Y=Lin_Pos.Y
N225_Short_Craft[Work_Area,4].Welding_Pos.Z=Lin_Pos.Z
N225_Short_Craft[Work_Area,4].Welding_Pos.A=Lin_Pos.A
N225_Short_Craft[Work_Area,4].Welding_Pos.B=Lin_Pos.B
N225_Short_Craft[Work_Area,4].Welding_Pos.C=Lin_Pos.C

ENDSWITCH


CASE #N315
;
SWITCH  Offset_No

CASE 1
SWITCH Sink_Welding_Size.Sink_Type
CASE #UpDown_One

Lin_Pos.X=D315_Start_POS.X
Lin_Pos.Y=D315_Start_POS.Y


;Lin_Pos.X=Sink_Welding_Size.Sink_Size_Width+Sink_Welding_Size.Sink_Size_Down_Distance*2
;Lin_Pos.Y=Sink_Welding_Size.Sink_Size_Short_OnePos+Sink_Welding_Size.Sink_Size_Short_TwoPos
Lin_Pos.Z=-150.000
Lin_Pos.A=0
Lin_Pos.B=0
Lin_Pos.C=0

case #LeftRight_One


Lin_Pos.X=D315_Start_POS.X
Lin_Pos.Y=D315_Start_POS.Y

;Lin_Pos.X=Sink_Welding_Size.Sink_Size_Short_OnePos+Sink_Welding_Size.Sink_Size_Short_TwoPos
;Lin_Pos.Y=Sink_Welding_Size.Sink_Size_Long+Sink_Welding_Size.Sink_Size_Left_Distance*2
Lin_Pos.Z=-150.000
Lin_Pos.A=0
Lin_Pos.B=0
Lin_Pos.C=0
ENDSWITCH


N315_Short_Craft[Work_Area,1].Welding_Pos.X=Lin_Pos.X
N315_Short_Craft[Work_Area,1].Welding_Pos.Y=Lin_Pos.Y
N315_Short_Craft[Work_Area,1].Welding_Pos.Z=Lin_Pos.Z
N315_Short_Craft[Work_Area,1].Welding_Pos.A=Lin_Pos.A
N315_Short_Craft[Work_Area,1].Welding_Pos.B=Lin_Pos.B
N315_Short_Craft[Work_Area,1].Welding_Pos.C=Lin_Pos.C

CASE 2
SWITCH Sink_Welding_Size.Sink_Type
CASE #UpDown_One

Lin_Pos.X=D315_Start_POS.X
Lin_Pos.Y=D315_Start_POS.Y

;Lin_Pos.X=Sink_Welding_Size.Sink_Size_Width+Sink_Welding_Size.Sink_Size_Down_Distance*2
;Lin_Pos.Y=Sink_Welding_Size.Sink_Size_Short_OnePos+Sink_Welding_Size.Sink_Size_Short_TwoPos
Lin_Pos.Z=0
Lin_Pos.A=0
Lin_Pos.B=0
Lin_Pos.C=0

case #LeftRight_One

Lin_Pos.X=D315_Start_POS.X
Lin_Pos.Y=D315_Start_POS.Y


;Lin_Pos.X=Sink_Welding_Size.Sink_Size_Short_OnePos+Sink_Welding_Size.Sink_Size_Short_TwoPos
;Lin_Pos.Y=Sink_Welding_Size.Sink_Size_Long+Sink_Welding_Size.Sink_Size_Left_Distance*2
Lin_Pos.Z=0
Lin_Pos.A=0
Lin_Pos.B=0
Lin_Pos.C=0
ENDSWITCH


N315_Short_Craft[Work_Area,2].Welding_Pos.X=Lin_Pos.X
N315_Short_Craft[Work_Area,2].Welding_Pos.Y=Lin_Pos.Y
N315_Short_Craft[Work_Area,2].Welding_Pos.Z=Lin_Pos.Z
N315_Short_Craft[Work_Area,2].Welding_Pos.A=Lin_Pos.A
N315_Short_Craft[Work_Area,2].Welding_Pos.B=Lin_Pos.B
N315_Short_Craft[Work_Area,2].Welding_Pos.C=Lin_Pos.C

CASE 3
SWITCH Sink_Welding_Size.Sink_Type
CASE #UpDown_One

Lin_Pos.X=D315_End_POS.X
Lin_Pos.Y=D315_End_POS.Y


;Lin_Pos.X=Sink_Welding_Size.Sink_Size_Width+Sink_Welding_Size.Sink_Size_Down_Distance*2-Sink_Welding_Size.Sink_Size_Short_Side
;Lin_Pos.Y=Sink_Welding_Size.Sink_Size_Short_OnePos+Sink_Welding_Size.Sink_Size_Short_TwoPos
Lin_Pos.Z=0
Lin_Pos.A=0
Lin_Pos.B=0
Lin_Pos.C=0

case #LeftRight_One

Lin_Pos.X=D315_End_POS.X
Lin_Pos.Y=D315_End_POS.Y

;Lin_Pos.X=Sink_Welding_Size.Sink_Size_Short_OnePos+Sink_Welding_Size.Sink_Size_Short_TwoPos
;Lin_Pos.Y=Sink_Welding_Size.Sink_Size_Long+Sink_Welding_Size.Sink_Size_Left_Distance*2-Sink_Welding_Size.Sink_Size_Short_Side
Lin_Pos.Z=0
Lin_Pos.A=0
Lin_Pos.B=0
Lin_Pos.C=0
ENDSWITCH


N315_Short_Craft[Work_Area,3].Welding_Pos.X=Lin_Pos.X
N315_Short_Craft[Work_Area,3].Welding_Pos.Y=Lin_Pos.Y
N315_Short_Craft[Work_Area,3].Welding_Pos.Z=Lin_Pos.Z
N315_Short_Craft[Work_Area,3].Welding_Pos.A=Lin_Pos.A
N315_Short_Craft[Work_Area,3].Welding_Pos.B=Lin_Pos.B
N315_Short_Craft[Work_Area,3].Welding_Pos.C=Lin_Pos.C

CASE 4
SWITCH Sink_Welding_Size.Sink_Type
CASE #UpDown_One


UL_Equation(D315_Start_POS,D315_End_POS,(Surr_Path*0.01),Sink_Welding_Size.Sink_Size_R,Lin_Pos)

;Lin_Pos.X=Sink_Welding_Size.Sink_Size_Width+Sink_Welding_Size.Sink_Size_Down_Distance+Sink_Welding_Size.Sink_Size_Short_Side*(Surr_Path/100)
;Lin_Pos.Y=Sink_Welding_Size.Sink_Size_Short_OnePos+Sink_Welding_Size.Sink_Size_Short_TwoPos
Lin_Pos.Z=-150.000
Lin_Pos.A=0
Lin_Pos.B=0
Lin_Pos.C=0

case #LeftRight_One

UL_Equation(D315_Start_POS,D315_End_POS,(Surr_Path*0.01),Sink_Welding_Size.Sink_Size_R,Lin_Pos)

;Lin_Pos.X=Sink_Welding_Size.Sink_Size_Short_OnePos+Sink_Welding_Size.Sink_Size_Short_TwoPos
;Lin_Pos.Y=Sink_Welding_Size.Sink_Size_Long+Sink_Welding_Size.Sink_Size_Left_Distance+Sink_Welding_Size.Sink_Size_Short_Side*(Surr_Path/100)
Lin_Pos.Z=-150.000
Lin_Pos.A=0
Lin_Pos.B=0
Lin_Pos.C=0
ENDSWITCH

N315_Short_Craft[Work_Area,4].Welding_Pos.X=Lin_Pos.X
N315_Short_Craft[Work_Area,4].Welding_Pos.Y=Lin_Pos.Y
N315_Short_Craft[Work_Area,4].Welding_Pos.Z=Lin_Pos.Z
N315_Short_Craft[Work_Area,4].Welding_Pos.A=Lin_Pos.A
N315_Short_Craft[Work_Area,4].Welding_Pos.B=Lin_Pos.B
N315_Short_Craft[Work_Area,4].Welding_Pos.C=Lin_Pos.C
ENDSWITCH


ENDSWITCH

SWITCH Pos_Type

CASE #L_LIN_POS,#C_LIN_POS




Lin_Pos.X=Lin_Pos.X+Offset_info.X
Lin_Pos.Y=Lin_Pos.Y+Offset_info.Y
Lin_Pos.Z=Lin_Pos.Z+Offset_info.Z



CASE #C_CIR_POS





Cir_Middle_POS.X=Cir_Middle_POS.X+Offset_info.X
Cir_Middle_POS.Y=Cir_Middle_POS.Y+Offset_info.Y
Cir_Middle_POS.Z=Cir_Middle_POS.Z+Offset_info.Z

Cir_END_POS.X=Cir_END_POS.X+Offset_cir_info.X
Cir_END_POS.Y=Cir_END_POS.Y+Offset_cir_info.Y
Cir_END_POS.Z=Cir_END_POS.Z+Offset_cir_info.Z

ENDSWITCH


END

GLOBAL DEF HanGao_Camera_Offset(Vision_Model:IN ,Calibration_Area:IN,Work_Camera:IN, OFFSET_POS:OUT)
DECL E6POS OFFSET_POS,Cam_45_POS,Cam_135_POS,Cam_225_POS,Cam_315_POS
DECL INT Calibration_Area,Work_Camera
DECL Surround_Welding_Type Sink_Size
DECL REAL T_X,T_Y,Q_X,Q_Y
DECL Vision_Model_Enum Vision_Model



switch Work_Camera

CASE 1

Sink_Size=N1_Sink_Data
Cam_45_POS=N1_Cam_45_POS
Cam_135_POS=N1_Cam_135_POS
Cam_225_POS=N1_Cam_225_POS
Cam_315_POS=N1_Cam_315_POS

CASE 2
Sink_Size=N2_Sink_Data
Cam_45_POS=N2_Cam_45_POS
Cam_135_POS=N2_Cam_135_POS
Cam_225_POS=N2_Cam_225_POS
Cam_315_POS=N2_Cam_315_POS

ENDSWITCH



SWITCH Calibration_Area

CASE 1


Q_Y=Camera_Calibration_Data.Sink_Size_Left_Distance-Sink_Size.Sink_Size_Left_Distance
Q_X=(Camera_Calibration_Data.Sink_Size_Down_Distance+Camera_Calibration_Data.Sink_Size_Width)-(Sink_Size.Sink_Size_Down_Distance+Sink_Size.Sink_Size_Width)

SWITCH Vision_Model

case #Calibration

IF (ABS(Q_Y)>=Vision_Scope ) OR (ABS(Q_X)>=Vision_Scope)THEN
OFFSET_POS.X=Cam_45_POS.X-Q_X
OFFSET_POS.Y=Cam_45_POS.Y-Q_Y
OFFSET_POS.Z=Cam_45_POS.Z
ELSE
OFFSET_POS.X=Cam_45_POS.X
OFFSET_POS.Y=Cam_45_POS.Y
OFFSET_POS.Z=Cam_45_POS.Z
ENDIF

ENDSWITCH

CASE 2


Q_Y=Camera_Calibration_Data.Sink_Size_Left_Distance-Sink_Size.Sink_Size_Left_Distance
Q_X=Camera_Calibration_Data.Sink_Size_Down_Distance-Sink_Size.Sink_Size_Down_Distance


SWITCH Vision_Model

case #Calibration
IF (ABS(Q_Y)>=Vision_Scope ) OR (ABS(Q_X)>=Vision_Scope)THEN
OFFSET_POS.X=Cam_135_POS.X-Q_X
OFFSET_POS.Y=Cam_135_POS.Y-Q_Y
OFFSET_POS.Z=Cam_135_POS.Z
ELSE
OFFSET_POS.X=Cam_135_POS.X
OFFSET_POS.Y=Cam_135_POS.Y
OFFSET_POS.Z=Cam_135_POS.Z
ENDIF

ENDSWITCH


CASE 3

Q_Y=(Camera_Calibration_Data.Sink_Size_Left_Distance+Camera_Calibration_Data.Sink_Size_Long)  -(Sink_Size.Sink_Size_Left_Distance+Sink_Size.Sink_Size_Long)
Q_X=Camera_Calibration_Data.Sink_Size_Down_Distance-Sink_Size.Sink_Size_Down_Distance

SWITCH Vision_Model

case #Calibration

IF (ABS(Q_Y)>=Vision_Scope ) OR (ABS(Q_X)>=Vision_Scope)THEN
OFFSET_POS.X=Cam_225_POS.X-Q_X
OFFSET_POS.Y=Cam_225_POS.Y-Q_Y
OFFSET_POS.Z=Cam_225_POS.Z
ELSE
OFFSET_POS.X=Cam_225_POS.X
OFFSET_POS.Y=Cam_225_POS.Y
OFFSET_POS.Z=Cam_225_POS.Z
ENDIF

ENDSWITCH


CASE 4

Q_Y=(Camera_Calibration_Data.Sink_Size_Left_Distance+Camera_Calibration_Data.Sink_Size_Long)-(Sink_Size.Sink_Size_Left_Distance+Sink_Size.Sink_Size_Long)
Q_X=(Camera_Calibration_Data.Sink_Size_Down_Distance+Camera_Calibration_Data.Sink_Size_Width)-(Sink_Size.Sink_Size_Down_Distance+Sink_Size.Sink_Size_Width)

SWITCH Vision_Model

case #Calibration
IF (ABS(Q_Y)>=Vision_Scope ) OR (ABS(Q_X)>=Vision_Scope)THEN
OFFSET_POS.X=Cam_315_POS.X-Q_X
OFFSET_POS.Y=Cam_315_POS.Y-Q_Y
OFFSET_POS.Z=Cam_315_POS.Z
ELSE
OFFSET_POS.X=Cam_315_POS.X
OFFSET_POS.Y=Cam_315_POS.Y
OFFSET_POS.Z=Cam_315_POS.Z
ENDIF

ENDSWITCH


ENDSWITCH


SWITCH Vision_Model

case #Find_Model
IF (ABS(Q_Y)>=Vision_Scope ) OR (ABS(Q_X)>=Vision_Scope)THEN
OFFSET_POS.X=OFFSET_POS.X-Q_X
OFFSET_POS.Y=OFFSET_POS.Y-Q_Y
ENDIF
ENDSWITCH





END


GLOBAL DEF HanGao_Calibration_Point(Calibration_POS:OUT,Calib_NO:IN)
DECL E6POS Calibration_POS
DECL INT Calib_NO



switch Global_Calib_Model

Case #New

Calibration_Point[Calib_NO]=Calibration_POS

Case #Add


Case #Text

Calibration_POS.X=Calibration_Text[Calib_NO].X
Calibration_POS.Y=Calibration_Text[Calib_NO].Y
endswitch


END

GLOBAL DEF HanGao_Camera_Sink_Pos(Calibration:IN,Work_Camera:IN)
DECL INT Calibration,Work_Camera
DECL BOOL User_Revise
DECL CHAR Meg_Str[1024]
DECL Surround_Welding_Type Sink_Size

 Meg_Str[]="This operation will overwrite the original data, whether to confirm?"
 ;Global_Messages_Dlg( Meg_Str[] ,User_Revise)
User_Revise=true





IF User_Revise==TRUE THEN


switch Work_Camera

CASE 1

Sink_Size=N1_Sink_Data
SWITCH Calibration

CASE 1
N1_Cam_45_POS=$POS_ACT
CASE 2
N1_Cam_135_POS=$POS_ACT
CASE 3
N1_Cam_225_POS=$POS_ACT
CASE 4
N1_Cam_315_POS=$POS_ACT
ENDSWITCH


CASE 2

Sink_Size=N2_Sink_Data
SWITCH Calibration

CASE 1
N2_Cam_45_POS=$POS_ACT
CASE 2
N2_Cam_135_POS=$POS_ACT
CASE 3
N2_Cam_225_POS=$POS_ACT
CASE 4
N2_Cam_315_POS=$POS_ACT
ENDSWITCH

ENDSWITCH



Camera_Calibration_Data=Sink_Size



else



halt

endif

END


GLOBAL DEF HanGao_Base_Calculate(POS_1:IN,POS_2:IN,POS_3:IN,POS_4:IN,G_BASE:IN,Angle_Area:IN)
DECL E6POS POS_1
DECL E6POS POS_2
DECL E6POS POS_3
DECL E6POS POS_4
DECL Work_Area_Enum Angle_Area
DECL REAL Direction_Deg,ATan_Deg
DECL INT G_BASE,OPFFSET
DECL Calculate_Lin_Const Lin_1_CONST
DECL Calculate_Lin_Const Lin_2_CONST
DECL POS Lin_Curss
DECL CHAR Meg_Str[1024]
DECL BOOL User_Revise
DECL State_t _State



OPFFSET=0
Lin_Curss={X 0, Y 0, Z 0, A 0,B 0,C 0}




Lin_1_CONST.A=POS_2.Y-POS_1.Y
Lin_1_CONST.B=POS_1.X-POS_2.X
Lin_1_CONST.C=POS_2.X*POS_1.Y-POS_1.X*POS_2.Y

Lin_2_CONST.A=POS_4.Y-POS_3.Y
Lin_2_CONST.B=POS_3.X-POS_4.X
Lin_2_CONST.C=POS_4.X*POS_3.Y-POS_3.X*POS_4.Y


Lin_Curss.X=(Lin_1_CONST.B*Lin_2_CONST.C-Lin_2_CONST.B*Lin_1_CONST.C)/(Lin_1_CONST.A*Lin_2_CONST.B-Lin_2_CONST.A*Lin_1_CONST.B)
Lin_Curss.Y=(Lin_2_CONST.A*Lin_1_CONST.C-Lin_1_CONST.A*Lin_2_CONST.C)/(Lin_2_CONST.B*Lin_1_CONST.A-Lin_1_CONST.B*Lin_2_CONST.A)
Lin_Curss.Z=POS_1.Z



SWITCH Angle_Area


CASE #A0

Direction_Deg=-180.000

IF Lin_Curss.X<>POS_4.X THEN

ATan_Deg=ATAN2(ABS(POS_4.x-Lin_Curss.x),ABS(POS_4.y-Lin_Curss.y))

IF POS_4.X-Lin_Curss.X<0 THEN
Lin_Curss.A=Direction_Deg+ATan_Deg
ENDIF

IF POS_4.X-Lin_Curss.X>0 THEN
Lin_Curss.A=Direction_Deg-ATan_Deg
ENDIF


ELSE

Lin_Curss.A=Direction_Deg

ENDIF

CASE #A90

Direction_Deg=90.000

IF Lin_Curss.Y<>POS_4.Y THEN

ATan_Deg=ATAN2(ABS(POS_4.Y-Lin_Curss.Y),ABS(POS_4.X-Lin_Curss.X))

IF POS_4.Y-Lin_Curss.Y<0 THEN
Lin_Curss.A=Direction_Deg-ATan_Deg
ENDIF

IF POS_4.Y-Lin_Curss.Y>0 THEN
Lin_Curss.A=Direction_Deg+ATan_Deg
ENDIF


ELSE

Lin_Curss.A=Direction_Deg

ENDIF




CASE #A270

Direction_Deg=-90.000

IF Lin_Curss.Y<>POS_4.Y THEN

ATan_Deg=ATAN2(ABS(POS_4.Y-Lin_Curss.Y),ABS(POS_4.X-Lin_Curss.X))

IF POS_4.Y-Lin_Curss.Y<0 THEN
Lin_Curss.A=Direction_Deg+ATan_Deg
ENDIF

IF POS_4.Y-Lin_Curss.Y>0 THEN
Lin_Curss.A=Direction_Deg-ATan_Deg
ENDIF


ELSE

Lin_Curss.A=Direction_Deg

ENDIF




ENDSWITCH










Lin_Curss.B=0
Lin_Curss.C=-180.000


SWRITE( Meg_Str[] , _State , OPFFSET , "New_BASE[%d]=X:%7.3F,Y:%7.3F,Z:%7.3F,A:%7.3F,B:%7.3F,C:%7.3F" , G_BASE ,Lin_Curss.X,Lin_Curss.Y,Lin_Curss.Z,Lin_Curss.A,Lin_Curss.B,Lin_Curss.C)


Global_Messages_Dlg( Meg_Str[] ,User_Revise)

IF User_Revise==TRUE THEN

IF G_BASE<>0  THEN

BASE_DATA[G_BASE].X=Lin_Curss.X
BASE_DATA[G_BASE].Y=Lin_Curss.Y
BASE_DATA[G_BASE].Z=Lin_Curss.Z
BASE_DATA[G_BASE].A=Lin_Curss.A
BASE_DATA[G_BASE].B=Lin_Curss.B
BASE_DATA[G_BASE].C=Lin_Curss.C

ENDIF

ENDIF


END



GLOBAL DEF Global_Messages_Dlg( Messsage_All[]:IN , User_S:OUT)

DECL KrlMsg_T msg
DECL KrlMsgPar_T Par[3]
DECL KrlmsgOpt_T opt
DECL KrlMsgDlgSK_T SK[7]
DECL INT nHandle,keynumber,OPFFSET
DECl BOOL User_S
DECL CHAR Messsage_All[]



msg={modul[] "HanGao" ,Nr 7}
msg.msg_txt[] = Messsage_All[]
SK[1]={sk_Type #value, sk_txt[] "Yes"}
SK[2]={sk_type #value, sk_txt[] "NO" }

nHandle= Set_KrlDlg( msg, par[],sk[],opt)

IF (nHandle>0) THEN

While (Exists_KrlDlg(nHandle,keynumber))
 wait sec 0.1
ENDWhile

SWITCH keynumber
   case 1
   User_S=true

   case 2
   User_S=false

ENDSWITCH










ENDIF


END


;Ax+By+C=0
GLOBAL DEF Lin_Equation (P1:IN,P2:IN,L_A:OUT,L_B:OUT,L_C:OUT)
DECL E6POS P1,P2
DECL REAL A,B,C,L_A,L_B,L_C
L_A=0.00
L_B=0.00
L_C=0.00



L_A=P2.Y-P1.Y
L_B=P1.X-P2.X
L_C=P2.X*P1.Y-P1.X*P2.Y




END



;y=kx+b
GLOBAL DEF Lin_Equation_LTk (A:IN,B:IN,C:IN,K_K:OUT,K_B:OUT)
DECL REAL A,B,C,K_K,K_B
K_K=0
K_B=0

K_K=-(a/b)
K_B=-(c/b)



END

;Point-User distance
GLOBAL DEF UL_Equation (UP1:IN,UP2:IN,U_DIS:IN,C_L:IN, Result_Pos_1:OUT)
DECL E6POS UP1,UP2,Result_Pos_1,L_S,L_E
DECL REAL L_Distance,L_DIS_1,L_DIS_2,U_DIS,R_X,R_Y,C_L



PP_Equation(UP1,UP2,L_DIS_1)

L_S.X=C_L*(UP2.X-UP1.X)/L_DIS_1+UP1.X
L_S.Y=C_L*(UP2.Y-UP1.Y)/L_DIS_1+UP1.Y

L_E.X=(L_DIS_1-C_L)*(UP2.X-UP1.X)/L_DIS_1+UP1.X
L_E.Y=(L_DIS_1-C_L)*(UP2.Y-UP1.Y)/L_DIS_1+UP1.Y

PP_Equation(L_S,L_E,L_DIS_2)


Result_Pos_1.X=L_DIS_2*U_DIS*(L_E.X-L_S.X)/L_DIS_2+L_S.X
Result_Pos_1.Y=L_DIS_2*U_DIS*(L_E.Y-L_S.Y)/L_DIS_2+L_S.Y


; IF U_DIS>1 THEN

; Result_Pos_1.X=U_DIS*(UP2.X-UP1.X)/L_DIS+UP1.X
; Result_Pos_1.Y=U_DIS*(UP2.Y-UP1.Y)/L_DIS+UP1.Y

; ELSE

; Result_Pos_1.X=L_DIS*U_DIS*(UP2.X-UP1.X)/L_DIS+UP1.X
; Result_Pos_1.Y=L_DIS*U_DIS*(UP2.Y-UP1.Y)/L_DIS+UP1.Y

; ENDIF





END



;Point-Point distance
GLOBAL DEF PP_Equation (PP1:IN,PP2:IN,L_Distance:OUT)
DECL E6POS PP1,PP2
DECL REAL L_Distance


L_Distance=0



L_Distance=SQRT((PP2.X-PP1.X)*(PP2.X-PP1.X)+(PP2.Y-PP1.Y)*(PP2.Y-PP1.Y))



END

--- Glode_HanGao.dat ---
&ACCESS RVO1
&REL 298
&PARAM EDITMASK = *
&PARAM TEMPLATE = C:\KRC\Roboter\Template\vorgabe
&PARAM DISKPATH = KRC:\R1\Program\HK
DEFDAT  glode_hangao PUBLIC




;--------DECL_Enum---------------
GLOBAL ENUM Sink_Type_Enum UpDown_One,LeftRight_One,LeftRight_Two,Null
GLOBAL ENUM Area_Enum L0,C45,L90,C135,L180,C225,L270,C315,N45,N135,N225,N315
GLOBAL ENUM Pos_Type_Enum C_LIN_POS,C_CIR_POS,L_LIN_POS
GLOBAL ENUM Work_Area_Enum A0,A90,A270
GLOBAL ENUM Vision_Model_Enum Calibration,Find_Model
;----------------------------------
;---DECL-STRUC-------------------------


GLOBAL STRUC Surround_Welding_Type BOOL Write_Status,REAL Sink_Size_Long,REAL Sink_Size_Width,REAL Sink_Size_R,REAL Sink_Size_Short_Side,REAL Sink_Size_Short_OnePos,REAL Sink_Size_Short_TwoPos,REAL Sink_Size_Pots_Thick,REAL Sink_Size_Panel_Thick,INT Sink_Model,REAL Sink_Size_Left_Distance,REAL Sink_Size_Down_Distance,Sink_Type_Enum Sink_Type
GLOBAL STRUC LSC_TOOL_TYP INT LSR_MAX_PWR,INT LSR_MIN_PWR,INT LSR_Prg,REAL SNSR_Prg,INT SNSR_State,REAL GAS_Pressure,INT LSR_Dly,INT GAS_Pre_Flow,INT GAS_Post_Flow
GLOBAL STRUC Offset_POS REAL X,REAL Y,REAL Z,REAL A,REAL B,REAL C
GLOBAL STRUC Offset_CIR REAL C_X,REAL C_Y,REAL C_Z,REAL C_A,REAL C_B,REAL C_C
GLOBAL STRUC Calculate_Lin_Const REAL A,REAL B,REAL C
GLOBAL STRUC Calibration_Sink_TYP REAL Long,REAL Width




GLOBAL STRUC Surr_Welding_Craft_Type CHAR Welding_Name[20],E6POS Welding_Pos,REAL Welding_Power,REAL Welding_Speed,REAL Welding_Angle,INT Welding_CDIS,INT Welding_ACC,Offset_POS Welding_Offset,Offset_CIR Welding_Offset_CIR





;-------------------------------------


;----------DECL_Value----------------------
DECL GLOBAL Surround_Welding_Type SW_DEFAULT={Sink_Size_Long 50.0000,Sink_Size_Width 345.000,Sink_Size_R 10.0000,Sink_Size_Pots_Thick 0.750000,Sink_Size_Panel_Thick 2.85000,Sink_Model 952154,Sink_Type #UpDown_One}
DECL GLOBAL LSC_TOOL_TYP LTDEFAULT={LSR_MAX_PWR 500,LSR_MIN_PWR 50,LSR_Prg 1,SNSR_Prg 1.00000,SNSR_State 0,GAS_Pressure 1.00000,LSR_Dly 100,GAS_Pre_Flow 0,GAS_Post_Flow 0}
DECL GLOBAL Offset_POS FFDEFAULT={X 0.0,Y 0.0,Z 0.0,A 0.0,B 0.0,C 0.0}
DECL GLOBAL Offset_CIR FCDEFAULT={C_X 0.0,C_Y 0.0,C_Z 0.0,C_A 0.0,C_B 0.0,C_C 0.0}
DECL GLOBAL E6POS PODEFAULT={X 0.0,Y 0.0,Z 0.0,A 0.0,B 0.0,C 0.0}


DECL GLOBAL Surround_Welding_Type Camera_Calibration_Data={Sink_Size_Long 632.000,Sink_Size_Width 352.000,Sink_Size_R 10.0000,Sink_Size_Short_Side 23.0000,Sink_Size_Short_OnePos 36.0000,Sink_Size_Short_TwoPos 328.000,Sink_Size_Pots_Thick 0.750000,Sink_Size_Panel_Thick 0.0,Sink_Model 952154,Sink_Size_Left_Distance 24.0000,Sink_Size_Down_Distance 24.0000,Sink_Type #LeftRight_One}

DECL GLOBAL E6POS N1_Cam_45_POS={X 1765.00,Y -1.00106740E-34,Z 1784.00,A 0.0,B 90.0000,C 3.24968513E-36}
DECL GLOBAL E6POS N1_Cam_135_POS={X 1765.00,Y -9.34353299E-23,Z 1784.00,A 0.0,B 90.0000,C 3.03311614E-24}
DECL GLOBAL E6POS N1_Cam_225_POS={X 1765.00,Y 5.47478833E-11,Z 1784.00,A 0.0,B 90.0000,C -6.59667199E-13}
DECL GLOBAL E6POS N1_Cam_315_POS={X 0.0,Y 0.0,A 0.0,B 0.0,C 0.0}

DECL GLOBAL E6POS N2_Cam_45_POS={X 293.122131,Y 89.9176636,Z -80.0293961,A 0.441927105,B -0.0416148715,C -0.0704164580,S 'B0010',T 'B1010',E1 0.0,E2 0.0,E3 0.0,E4 0.0,E5 0.0,E6 0.0}
DECL GLOBAL E6POS N2_Cam_135_POS={X -42.3839874,Y 91.8151550,Z -80.0254822,A 0.441927105,B -0.0416148864,C -0.0704164430,S 'B0010',T 'B1010',E1 0.0,E2 0.0,E3 0.0,E4 0.0,E5 0.0,E6 0.0}
DECL GLOBAL E6POS N2_Cam_225_POS={X -39.7999954,Y 716.082336,Z -80.0293350,A 0.441926539,B -0.0416153781,C -0.0704161152,S 'B0010',T 'B00101011',E1 0.0,E2 0.0,E3 0.0,E4 0.0,E5 0.0,E6 0.0}
DECL GLOBAL E6POS N2_Cam_315_POS={X 294.984924,Y 714.198059,Z -80.0293350,A 0.441925645,B -0.0416159667,C -0.0704158247,S 'B0010',T 'B00101011',E1 0.0,E2 0.0,E3 0.0,E4 0.0,E5 0.0,E6 0.0}

DECL GLOBAL E6POS N45_OFFSET_POS={X 375.675,Y 23.4770,Z 0.0,A 0.0,B 0.0,C 0.0}
DECL GLOBAL E6POS N135_OFFSET_POS={X 24.0190,Y 23.1910,Z 0.0,A 0.0,B 0.0,C 0.0}
DECL GLOBAL E6POS N225_OFFSET_POS={X 23.4020,Y 725.222,Z 0.0,A 0.0,B 0.0,C 0.0}
DECL GLOBAL E6POS N315_OFFSET_POS={X 375.730,Y 725.747,Z 0.0,A 0.0,B 0.0,C 0.0}

DECL GLOBAL E6POS N45_CIR_POS={X 372.590,Y 27.2660,Z 0.0,A 0.0,B 0.0,C 0.0}
DECL GLOBAL E6POS N135_CIR_POS={X 27.7730,Y 26.2530,Z 0.0,A 0.0,B 0.0,C 0.0}
DECL GLOBAL E6POS N225_CIR_POS={X 27.3020,Y 722.048,Z 0.0,A 0.0,B 0.0,C 0.0}
DECL GLOBAL E6POS N315_CIR_POS={X 372.023,Y 722.369,Z 0.0,A 0.0,B 0.0,C 0.0}

DECL GLOBAL E6POS D45_Start_POS={X 364.343,Y -0.734000,Z 0.0,A 0.0,B 0.0,C 0.0}
DECL GLOBAL E6POS D45_End_POS={X 364.315,Y 23.5880,Z 0.0,A 0.0,B 0.0,C 0.0}
DECL GLOBAL E6POS D135_Start_POS={X 37.1160,Y -1.02700,Z 0.0,A 0.0,B 0.0,C 0.0}
DECL GLOBAL E6POS D135_End_POS={X 37.2780,Y 23.2150,Z 0.0,A 0.0,B 0.0,C 0.0}
DECL GLOBAL E6POS D225_Start_POS={X 36.7810,Y 749.275,Z 0.0,A 0.0,B 0.0,C 0.0}
DECL GLOBAL E6POS D225_End_POS={X 36.9310,Y 725.260,Z 0.0,A 0.0,B 0.0,C 0.0}
DECL GLOBAL E6POS D315_Start_POS={X 364.063,Y 750.089,Z 0.0,A 0.0,B 0.0,C 0.0}
DECL GLOBAL E6POS D315_End_POS={X 364.380,Y 725.694,Z 0.0,A 0.0,B 0.0,C 0.0}


DECL GLOBAL Surr_Welding_Craft_Type L0_Welding_Craft[2,10]
L0_Welding_Craft[1,1]={Welding_Name[] "S2",Welding_Pos {X 120.000,Y 38.0000,Z 0.0,A 0.0,B 20.0000,C 0.0},Welding_Power 80.0000,Welding_Speed 0.0400000,Welding_Angle 20.0000,Welding_CDIS 5,Welding_ACC 100,Welding_Offset {X 0.0,Y 0.0,Z 0.0}}
L0_Welding_Craft[1,2]={Welding_Name[] "L0_S2",Welding_Pos {X 376.000,Y 584.800,Z 0.0,A 0.0,B 20.0000,C 0.0},Welding_Power 80.0000,Welding_Speed 0.0400000,Welding_Angle 20.0000,Welding_CDIS 5,Welding_ACC 100,Welding_Offset {X 0.0,Y 0.0,Z 0.0}}
L0_Welding_Craft[1,3]={Welding_Name[] "L0_S3",Welding_Pos {X 376.000,Y 340.000,Z 0.0,A 0.0,B 20.0000,C 0.0},Welding_Power 80.0000,Welding_Speed 0.0400000,Welding_Angle 20.0000,Welding_CDIS 5,Welding_ACC 100,Welding_Offset {X 0.0,Y 0.0,Z 0.0}}
L0_Welding_Craft[1,4]={Welding_Name[] "L0_S4",Welding_Pos {X 376.000,Y 64.6000061,Z 0.0,A 0.0,B 20.0000,C 0.0},Welding_Power 80.0000,Welding_Speed 0.0400000,Welding_Angle 20.0000,Welding_CDIS 5,Welding_ACC 100,Welding_Offset {X 0.0,Y 0.0,Z 0.0}}
L0_Welding_Craft[1,5]={Welding_Name[] "S1",Welding_Pos {X 400.000,Y 86.0000153,Z -3.00000,A 0.0,B 23.0000,C 0.0},Welding_Power 80.0000,Welding_Speed 0.0400000,Welding_Angle 20.0000,Welding_CDIS 5,Welding_ACC 100,Welding_Offset {X 0.0,Y 0.0,Z 0.0}}
L0_Welding_Craft[1,6]={Welding_Name[] "S6",Welding_Pos {X 533.000,Y 463.600037,Z -2.05000,A 0.0,B -23.0000,C 0.0},Welding_Power 80.0000,Welding_Speed 0.0400000,Welding_Angle 20.0000,Welding_CDIS 5,Welding_ACC 100,Welding_Offset {X 0.0,Y 0.0,Z 0.0}}
L0_Welding_Craft[1,7]={Welding_Name[] "S7",Welding_Pos {X 533.000,Y 463.600037,Z -2.05000,A 0.0,B -23.0000,C 0.0},Welding_Power 80.0000,Welding_Speed 0.0400000,Welding_Angle 20.0000,Welding_CDIS 5,Welding_ACC 100,Welding_Offset {X 0.0,Y 0.0,Z 0.0}}
L0_Welding_Craft[1,8]={Welding_Name[] "S8",Welding_Pos {X 533.000,Y 463.600037,Z -2.05000,A 0.0,B -23.0000,C 0.0},Welding_Power 80.0000,Welding_Speed 0.0400000,Welding_Angle 20.0000,Welding_CDIS 5,Welding_ACC 100,Welding_Offset {X 0.0,Y 0.0,Z 0.0}}
L0_Welding_Craft[1,9]={Welding_Name[] "S9",Welding_Pos {X 533.000,Y 463.600037,Z -2.05000,A 0.0,B -23.0000,C 0.0},Welding_Power 80.0000,Welding_Speed 0.0400000,Welding_Angle 20.0000,Welding_CDIS 5,Welding_ACC 100,Welding_Offset {X 0.0,Y 0.0,Z 0.0}}
L0_Welding_Craft[1,10]={Welding_Name[] "S10",Welding_Pos {X 533.000,Y 338.000,Z -2.05000,A 0.0,B -23.0000,C 0.0},Welding_Power 80.0000,Welding_Speed 0.0400000,Welding_Angle 20.0000,Welding_CDIS 5,Welding_ACC 100,Welding_Offset {X 0.0,Y 0.0,Z 0.0}}
L0_Welding_Craft[2,1]={Welding_Name[] "L0_S1",Welding_Pos {X 375.681122,Y 101.703979,Z 0.0,A 0.0,B 20.0000,C 0.0},Welding_Power 80.0000,Welding_Speed 0.300000,Welding_Angle 20.0000,Welding_CDIS 5,Welding_ACC 100,Welding_Offset {X 0.0,Y 0.0,Z 0.0}}
L0_Welding_Craft[2,2]={Welding_Name[] "L0_S2",Welding_Pos {X 375.566071,Y 647.351257,Z 0.0,A 0.0,B 20.0000,C 0.0},Welding_Power 80.0000,Welding_Speed 0.0320000,Welding_Angle 20.0000,Welding_CDIS 5,Welding_ACC 100,Welding_Offset {X 0.0,Y -1.50000,Z 0.0}}
L0_Welding_Craft[2,3]={Welding_Name[] "L0_S3",Welding_Pos {X 375.650,Y 374.428497,Z 0.0,A 0.0,B 20.0000,C 0.0},Welding_Power 80.0000,Welding_Speed 0.0320000,Welding_Angle 20.0000,Welding_CDIS 5,Welding_ACC 100,Welding_Offset {X 0.0,Y -1.80000,Z 0.0}}
L0_Welding_Craft[2,4]={Welding_Name[] "L0_S4",Welding_Pos {X 375.744415,Y 67.3903809,Z 0.0,A 0.0,B 20.0000,C 0.0},Welding_Power 80.0000,Welding_Speed 0.0340000,Welding_Angle 20.0000,Welding_CDIS 5,Welding_ACC 100,Welding_Offset {X 0.0,Y -1.00000,Z 0.0}}
L0_Welding_Craft[2,5]={Welding_Name[] "S1",Welding_Pos {X 400.000,Y 86.0000153,Z -3.00000,A 0.0,B 23.0000,C 0.0},Welding_Power 80.0000,Welding_Speed 0.0400000,Welding_Angle 20.0000,Welding_CDIS 5,Welding_ACC 100,Welding_Offset {X 0.0,Y 0.0,Z 0.0}}
L0_Welding_Craft[2,6]={Welding_Name[] "S6",Welding_Pos {X 533.000,Y 463.600037,Z -2.05000,A 0.0,B -23.0000,C 0.0},Welding_Power 80.0000,Welding_Speed 0.0400000,Welding_Angle 20.0000,Welding_CDIS 5,Welding_ACC 100,Welding_Offset {X 0.0,Y 0.0,Z 0.0}}
L0_Welding_Craft[2,7]={Welding_Name[] "S7",Welding_Pos {X 533.000,Y 463.600037,Z -2.05000,A 0.0,B -23.0000,C 0.0},Welding_Power 80.0000,Welding_Speed 0.0400000,Welding_Angle 20.0000,Welding_CDIS 5,Welding_ACC 100,Welding_Offset {X 0.0,Y 0.0,Z 0.0}}
L0_Welding_Craft[2,8]={Welding_Name[] "S8",Welding_Pos {X 533.000,Y 463.600037,Z -2.05000,A 0.0,B -23.0000,C 0.0},Welding_Power 80.0000,Welding_Speed 0.0400000,Welding_Angle 20.0000,Welding_CDIS 5,Welding_ACC 100,Welding_Offset {X 0.0,Y 0.0,Z 0.0}}
L0_Welding_Craft[2,9]={Welding_Name[] "S9",Welding_Pos {X 533.000,Y 463.600037,Z -2.05000,A 0.0,B -23.0000,C 0.0},Welding_Power 80.0000,Welding_Speed 0.0400000,Welding_Angle 20.0000,Welding_CDIS 5,Welding_ACC 100,Welding_Offset {X 0.0,Y 0.0,Z 0.0}}
L0_Welding_Craft[2,10]={Welding_Name[] "S10",Welding_Pos {X 533.000,Y 338.000,Z -2.05000,A 0.0,B -23.0000,C 0.0},Welding_Power 80.0000,Welding_Speed 0.0400000,Welding_Angle 20.0000,Welding_CDIS 5,Welding_ACC 100,Welding_Offset {X 0.0,Y 0.0,Z 0.0}}



DECL GLOBAL Surr_Welding_Craft_Type C45_Welding_Craft[2,3]
C45_Welding_Craft[1,1]={Welding_Name[] "S3",Welding_Pos {X 120.000,Y 30.0000,Z 0.0,A 0.0,B 20.0000,C 0.0},Welding_Power 80.0000,Welding_Speed 0.0400000,Welding_Angle 20.0000,Welding_CDIS 5,Welding_ACC 100,Welding_Offset {X 0.0,Y 0.0,Z 0.0}}
C45_Welding_Craft[1,2]={Welding_Name[] "PM2",Welding_Pos {X 117.070,Y 22.9300,Z 0.0,A 0.0,B 0.0,C 0.0},Welding_Power 80.0000,Welding_Speed 0.0400000,Welding_Angle 20.0000,Welding_CDIS 5,Welding_ACC 100,Welding_Offset {X 0.0,Y 0.0,Z 0.0},Welding_Offset_CIR {C_X 0.0,C_Y 0.0,C_Z 0.0}}
C45_Welding_Craft[1,3]={Welding_Name[] "PE2",Welding_Pos {X 110.000,Y 20.0000,Z 0.0,A 0.0,B 0.0,C 20.0000},Welding_Power 80.0000,Welding_Speed 0.0400000,Welding_Angle 20.0000,Welding_CDIS 5,Welding_ACC 100,Welding_Offset {X 0.0,Y 0.0,Z 0.0}}
C45_Welding_Craft[2,1]={Welding_Name[] "C45_S1",Welding_Pos {X 375.754913,Y 33.2750244,Z 0.0,A 0.0,B 20.0000,C 0.0},Welding_Power 80.0000,Welding_Speed 0.0300000,Welding_Angle 20.0000,Welding_CDIS 5,Welding_ACC 100,Welding_Offset {X 0.0,Y 0.0,Z 0.0}}
C45_Welding_Craft[2,2]={Welding_Name[] "PM3",Welding_Pos {X 372.649,Y 27.0560,Z 0.0,A 0.0,B 0.0,C 0.0},Welding_Power 80.0000,Welding_Speed 0.0400000,Welding_Angle 20.0000,Welding_CDIS 5,Welding_ACC 100,Welding_Offset {X 0.0,Y 0.500000,Z 0.0},Welding_Offset_CIR {C_X 0.0,C_Y 0.0,C_Z 0.0}}
C45_Welding_Craft[2,3]={Welding_Name[] "PE3",Welding_Pos {X 365.758,Y 23.2745743,Z 0.0,A 0.0,B 0.0,C 20.0000},Welding_Power 80.0000,Welding_Speed 0.0120000,Welding_Angle 20.0000,Welding_CDIS 5,Welding_ACC 100,Welding_Offset {X 0.0,Y 0.500000,Z 0.0}}


DECL GLOBAL Surr_Welding_Craft_Type L90_Welding_Craft[2,10]
L90_Welding_Craft[1,1]={Welding_Name[] "S2",Welding_Pos {X 30.0000,Y 20.0000,Z 0.0,A 0.0,B 0.0,C 20.0000},Welding_Power 80.0000,Welding_Speed 0.0400000,Welding_Angle 20.0000,Welding_CDIS 5,Welding_ACC 100,Welding_Offset {X 0.0,Y 0.0,Z 0.0}}
L90_Welding_Craft[1,2]={Welding_Name[] "L90_S2",Welding_Pos {X 200.000,Y 24.0000,Z 0.0,A 0.0,B 0.0,C 20.0000},Welding_Power 80.0000,Welding_Speed 0.0400000,Welding_Angle 20.0000,Welding_CDIS 5,Welding_ACC 100,Welding_Offset {X 0.0,Y 0.0,Z 0.0}}
L90_Welding_Craft[1,3]={Welding_Name[] "L90_S3",Welding_Pos {X 67.2000122,Y 24.0000,Z 0.0,A 0.0,B 0.0,C 20.0000},Welding_Power 80.0000,Welding_Speed 0.0400000,Welding_Angle 20.0000,Welding_CDIS 5,Welding_ACC 100,Welding_Offset {X 0.0,Y 0.0,Z 0.0}}
L90_Welding_Craft[1,4]={Welding_Name[] "S4",Welding_Pos {X 400.000,Y 86.0000153,Z -3.00000,A 0.0,B 23.0000,C 0.0},Welding_Power 80.0000,Welding_Speed 0.0400000,Welding_Angle 20.0000,Welding_CDIS 5,Welding_ACC 100,Welding_Offset {X 0.0,Y 0.0,Z 0.0}}
L90_Welding_Craft[1,5]={Welding_Name[] "S5",Welding_Pos {X 371.000,Y 0.0,Z -3.00000,A 0.0,B 0.0,C 23.0000},Welding_Power 80.0000,Welding_Speed 0.0400000,Welding_Angle 20.0000,Welding_CDIS 5,Welding_ACC 100,Welding_Offset {X 0.0,Y 0.0,Z 0.0}}
L90_Welding_Craft[1,6]={Welding_Name[] "S6",Welding_Pos {X 533.000,Y 463.600037,Z -2.05000,A 0.0,B -23.0000,C 0.0},Welding_Power 80.0000,Welding_Speed 0.0400000,Welding_Angle 20.0000,Welding_CDIS 5,Welding_ACC 100,Welding_Offset {X 0.0,Y 0.0,Z 0.0}}
L90_Welding_Craft[1,7]={Welding_Name[] "S7",Welding_Pos {X 533.000,Y 463.600037,Z -2.05000,A 0.0,B -23.0000,C 0.0},Welding_Power 80.0000,Welding_Speed 0.0400000,Welding_Angle 20.0000,Welding_CDIS 5,Welding_ACC 100,Welding_Offset {X 0.0,Y 0.0,Z 0.0}}
L90_Welding_Craft[1,8]={Welding_Name[] "S8",Welding_Pos {X 533.000,Y 463.600037,Z -2.05000,A 0.0,B -23.0000,C 0.0},Welding_Power 80.0000,Welding_Speed 0.0400000,Welding_Angle 20.0000,Welding_CDIS 5,Welding_ACC 100,Welding_Offset {X 0.0,Y 0.0,Z 0.0}}
L90_Welding_Craft[1,9]={Welding_Name[] "S9",Welding_Pos {X 533.000,Y 463.600037,Z -2.05000,A 0.0,B -23.0000,C 0.0},Welding_Power 80.0000,Welding_Speed 0.0400000,Welding_Angle 20.0000,Welding_CDIS 5,Welding_ACC 100,Welding_Offset {X 0.0,Y 0.0,Z 0.0}}
L90_Welding_Craft[1,10]={Welding_Name[] "S10",Welding_Pos {X 533.000,Y 338.000,Z -2.05000,A 0.0,B -23.0000,C 0.0},Welding_Power 80.0000,Welding_Speed 0.0400000,Welding_Angle 20.0000,Welding_CDIS 5,Welding_ACC 100,Welding_Offset {X 0.0,Y 0.0,Z 0.0}}
L90_Welding_Craft[2,1]={Welding_Name[] "L90_S1",Welding_Pos {X 332.548584,Y 23.2731590,Z 0.0,A 0.0,B 0.0,C 20.0000},Welding_Power 80.0000,Welding_Speed 0.0320000,Welding_Angle 20.0000,Welding_CDIS 5,Welding_ACC 100,Welding_Offset {X 0.0,Y 0.800000,Z 0.0}}
L90_Welding_Craft[2,2]={Welding_Name[] "L90_S2",Welding_Pos {X 199.711,Y 23.2675,Z 0.0,A 0.0,B 0.0,C 20.0000},Welding_Power 80.0000,Welding_Speed 0.0320000,Welding_Angle 20.0000,Welding_CDIS 5,Welding_ACC 100,Welding_Offset {X 0.0,Y 0.800000,Z 0.0}}
L90_Welding_Craft[2,3]={Welding_Name[] "L90_S3",Welding_Pos {X 66.8734131,Y 23.2618408,Z 0.0,A 0.0,B 0.0,C 20.0000},Welding_Power 80.0000,Welding_Speed 0.0320000,Welding_Angle 20.0000,Welding_CDIS 5,Welding_ACC 100,Welding_Offset {X 0.0,Y 0.800000,Z 0.0}}
L90_Welding_Craft[2,4]={Welding_Name[] "S4",Welding_Pos {X 400.000,Y 86.0000153,Z -3.00000,A 0.0,B 23.0000,C 0.0},Welding_Power 80.0000,Welding_Speed 0.0400000,Welding_Angle 20.0000,Welding_CDIS 5,Welding_ACC 100,Welding_Offset {X 0.0,Y 0.0,Z 0.0}}
L90_Welding_Craft[2,5]={Welding_Name[] "S5",Welding_Pos {X 371.000,Y 0.0,Z -3.00000,A 0.0,B 0.0,C 23.0000},Welding_Power 80.0000,Welding_Speed 0.0400000,Welding_Angle 20.0000,Welding_CDIS 5,Welding_ACC 100,Welding_Offset {X 0.0,Y 0.0,Z 0.0}}
L90_Welding_Craft[2,6]={Welding_Name[] "S6",Welding_Pos {X 533.000,Y 463.600037,Z -2.05000,A 0.0,B -23.0000,C 0.0},Welding_Power 80.0000,Welding_Speed 0.0400000,Welding_Angle 20.0000,Welding_CDIS 5,Welding_ACC 100,Welding_Offset {X 0.0,Y 0.0,Z 0.0}}
L90_Welding_Craft[2,7]={Welding_Name[] "S7",Welding_Pos {X 533.000,Y 463.600037,Z -2.05000,A 0.0,B -23.0000,C 0.0},Welding_Power 80.0000,Welding_Speed 0.0400000,Welding_Angle 20.0000,Welding_CDIS 5,Welding_ACC 100,Welding_Offset {X 0.0,Y 0.0,Z 0.0}}
L90_Welding_Craft[2,8]={Welding_Name[] "S8",Welding_Pos {X 533.000,Y 463.600037,Z -2.05000,A 0.0,B -23.0000,C 0.0},Welding_Power 80.0000,Welding_Speed 0.0400000,Welding_Angle 20.0000,Welding_CDIS 5,Welding_ACC 100,Welding_Offset {X 0.0,Y 0.0,Z 0.0}}
L90_Welding_Craft[2,9]={Welding_Name[] "S9",Welding_Pos {X 533.000,Y 463.600037,Z -2.05000,A 0.0,B -23.0000,C 0.0},Welding_Power 80.0000,Welding_Speed 0.0400000,Welding_Angle 20.0000,Welding_CDIS 5,Welding_ACC 100,Welding_Offset {X 0.0,Y 0.0,Z 0.0}}
L90_Welding_Craft[2,10]={Welding_Name[] "S10",Welding_Pos {X 533.000,Y 338.000,Z -2.05000,A 0.0,B -23.0000,C 0.0},Welding_Power 80.0000,Welding_Speed 0.0400000,Welding_Angle 20.0000,Welding_CDIS 5,Welding_ACC 100,Welding_Offset {X 0.0,Y 0.0,Z 0.0}}

DECL GLOBAL Surr_Welding_Craft_Type C135_Welding_Craft[2,3]
C135_Welding_Craft[1,1]={Welding_Name[] "S3",Welding_Pos {X 30.0000,Y 20.0000,Z 0.0,A 0.0,B 0.0,C 20.0000},Welding_Power 80.0000,Welding_Speed 0.0400000,Welding_Angle 20.0000,Welding_CDIS 5,Welding_ACC 100,Welding_Offset {X 0.0,Y 0.0,Z 0.0}}
C135_Welding_Craft[1,2]={Welding_Name[] "PM3",Welding_Pos {X 22.9300,Y 22.9300,Z 0.0,A 0.0,B 0.0,C 0.0},Welding_Power 80.0000,Welding_Speed 0.0400000,Welding_Angle -20.0000,Welding_CDIS 5,Welding_ACC 100,Welding_Offset {X 0.0,Y 0.0,Z 0.0},Welding_Offset_CIR {C_X 0.0,C_Y 0.0,C_Z 0.0}}
C135_Welding_Craft[1,3]={Welding_Name[] "PE3",Welding_Pos {X 20.0000,Y 30.0000,Z 0.0,A 0.0,B -20.0000,C 0.0},Welding_Power 80.0000,Welding_Speed 0.0400000,Welding_Angle -20.0000,Welding_CDIS 5,Welding_ACC 100,Welding_Offset {X 0.0,Y 0.0,Z 0.0}}
C135_Welding_Craft[2,1]={Welding_Name[] "C135_S1",Welding_Pos {X 33.6640,Y 23.2604256,Z 0.0,A 0.0,B 0.0,C 20.0000},Welding_Power 80.0000,Welding_Speed 0.0300000,Welding_Angle 20.0000,Welding_CDIS 5,Welding_ACC 100,Welding_Offset {X 0.0,Y 0.500000,Z 0.0}}
C135_Welding_Craft[2,2]={Welding_Name[] "PM4",Welding_Pos {X 27.4390,Y 26.3430,Z 0.0,A 0.0,B 0.0,C 0.0},Welding_Power 80.0000,Welding_Speed 0.0400000,Welding_Angle -20.0000,Welding_CDIS 5,Welding_ACC 100,Welding_Offset {X 0.0,Y 0.0,Z 0.0},Welding_Offset_CIR {C_X 0.0,C_Y 0.0,C_Z 0.0}}
C135_Welding_Craft[2,3]={Welding_Name[] "PE4",Welding_Pos {X 23.6575489,Y 33.2600,Z 0.0,A 0.0,B -20.0000,C 0.0},Welding_Power 80.0000,Welding_Speed 0.0150000,Welding_Angle -20.0000,Welding_CDIS 5,Welding_ACC 100,Welding_Offset {X 0.0,Y 0.500000,Z 0.0}}

DECL GLOBAL Surr_Welding_Craft_Type L180_Welding_Craft[2,10]
L180_Welding_Craft[1,1]={Welding_Name[] "S2",Welding_Pos {X 20.0000,Y 30.0000,Z 0.0,A 0.0,B -20.0000,C 0.0},Welding_Power 80.0000,Welding_Speed 0.0400000,Welding_Angle -20.0000,Welding_CDIS 5,Welding_ACC 100,Welding_Offset {X 0.0,Y 0.0,Z 0.0}}
L180_Welding_Craft[1,2]={Welding_Name[] "L180_S2",Welding_Pos {X 24.0000,Y 340.000,Z 0.0,A 0.0,B -20.0000,C 0.0},Welding_Power 80.0000,Welding_Speed 0.0400000,Welding_Angle -20.0000,Welding_CDIS 5,Welding_ACC 100,Welding_Offset {X 0.0,Y 0.0,Z 0.0}}
L180_Welding_Craft[1,3]={Welding_Name[] "L180_S3",Welding_Pos {X 24.0000,Y 615.399963,Z 0.0,A 0.0,B -20.0000,C 0.0},Welding_Power 80.0000,Welding_Speed 0.0400000,Welding_Angle -20.0000,Welding_CDIS 5,Welding_ACC 100,Welding_Offset {X 0.0,Y 0.0,Z 0.0}}
L180_Welding_Craft[1,4]={Welding_Name[] "S4",Welding_Pos {X 400.000,Y 86.0000153,Z -3.00000,A 0.0,B 23.0000,C 0.0},Welding_Power 80.0000,Welding_Speed 0.0400000,Welding_Angle -20.0000,Welding_CDIS 5,Welding_ACC 100,Welding_Offset {X 0.0,Y 0.0,Z 0.0}}
L180_Welding_Craft[1,5]={Welding_Name[] "S5",Welding_Pos {X 0.0,Y 371.000,Z -3.00000,A 0.0,B -23.0000,C 0.0},Welding_Power 80.0000,Welding_Speed 0.0400000,Welding_Angle -20.0000,Welding_CDIS 5,Welding_ACC 100,Welding_Offset {X 0.0,Y 0.0,Z 0.0}}
L180_Welding_Craft[1,6]={Welding_Name[] "S6",Welding_Pos {X 533.000,Y 463.600037,Z -2.05000,A 0.0,B -23.0000,C 0.0},Welding_Power 80.0000,Welding_Speed 0.0400000,Welding_Angle -20.0000,Welding_CDIS 5,Welding_ACC 100,Welding_Offset {X 0.0,Y 0.0,Z 0.0}}
L180_Welding_Craft[1,7]={Welding_Name[] "S7",Welding_Pos {X 533.000,Y 463.600037,Z -2.05000,A 0.0,B -23.0000,C 0.0},Welding_Power 80.0000,Welding_Speed 0.0400000,Welding_Angle -20.0000,Welding_CDIS 5,Welding_ACC 100,Welding_Offset {X 0.0,Y 0.0,Z 0.0}}
L180_Welding_Craft[1,8]={Welding_Name[] "S8",Welding_Pos {X 533.000,Y 463.600037,Z -2.05000,A 0.0,B -23.0000,C 0.0},Welding_Power 80.0000,Welding_Speed 0.0400000,Welding_Angle -20.0000,Welding_CDIS 5,Welding_ACC 100,Welding_Offset {X 0.0,Y 0.0,Z 0.0}}
L180_Welding_Craft[1,9]={Welding_Name[] "S9",Welding_Pos {X 533.000,Y 463.600037,Z -2.05000,A 0.0,B -23.0000,C 0.0},Welding_Power 80.0000,Welding_Speed 0.0400000,Welding_Angle -20.0000,Welding_CDIS 5,Welding_ACC 100,Welding_Offset {X 0.0,Y 0.0,Z 0.0}}
L180_Welding_Craft[1,10]={Welding_Name[] "S10",Welding_Pos {X 533.000,Y 338.000,Z -2.05000,A 0.0,B -23.0000,C 0.0},Welding_Power 80.0000,Welding_Speed 0.0400000,Welding_Angle -20.0000,Welding_CDIS 5,Welding_ACC 100,Welding_Offset {X 0.0,Y 0.0,Z 0.0}}
L180_Welding_Craft[2,1]={Welding_Name[] "L180_S1",Welding_Pos {X 23.6135387,Y 101.477905,Z 0.0,A 0.0,B -20.0000,C 0.0},Welding_Power 80.0000,Welding_Speed 0.0320000,Welding_Angle -20.0000,Welding_CDIS 5,Welding_ACC 100,Welding_Offset {X 0.0,Y 0.0,Z 0.0}}
L180_Welding_Craft[2,2]={Welding_Name[] "L180_S2",Welding_Pos {X 23.4375,Y 374.349518,Z 0.0,A 0.0,B -20.0000,C 0.0},Welding_Power 80.0000,Welding_Speed 0.0320000,Welding_Angle -20.0000,Welding_CDIS 5,Welding_ACC 100,Welding_Offset {X 0.0,Y 0.0,Z 0.0}}
L180_Welding_Craft[2,3]={Welding_Name[] "L180_S3",Welding_Pos {X 23.2394562,Y 681.330078,Z 0.0,A 0.0,B -20.0000,C 0.0},Welding_Power 80.0000,Welding_Speed 0.0320000,Welding_Angle -20.0000,Welding_CDIS 5,Welding_ACC 100,Welding_Offset {X 0.200000,Y 0.0,Z 0.0}}
L180_Welding_Craft[2,4]={Welding_Name[] "S4",Welding_Pos {X 400.000,Y 86.0000153,Z -3.00000,A 0.0,B 23.0000,C 0.0},Welding_Power 80.0000,Welding_Speed 0.0400000,Welding_Angle -20.0000,Welding_CDIS 5,Welding_ACC 100,Welding_Offset {X 0.0,Y 0.0,Z 0.0}}
L180_Welding_Craft[2,5]={Welding_Name[] "S5",Welding_Pos {X 0.0,Y 371.000,Z -3.00000,A 0.0,B -23.0000,C 0.0},Welding_Power 80.0000,Welding_Speed 0.0400000,Welding_Angle -20.0000,Welding_CDIS 5,Welding_ACC 100,Welding_Offset {X 0.0,Y 0.0,Z 0.0}}
L180_Welding_Craft[2,6]={Welding_Name[] "S6",Welding_Pos {X 533.000,Y 463.600037,Z -2.05000,A 0.0,B -23.0000,C 0.0},Welding_Power 80.0000,Welding_Speed 0.0400000,Welding_Angle -20.0000,Welding_CDIS 5,Welding_ACC 100,Welding_Offset {X 0.0,Y 0.0,Z 0.0}}
L180_Welding_Craft[2,7]={Welding_Name[] "S7",Welding_Pos {X 533.000,Y 463.600037,Z -2.05000,A 0.0,B -23.0000,C 0.0},Welding_Power 80.0000,Welding_Speed 0.0400000,Welding_Angle -20.0000,Welding_CDIS 5,Welding_ACC 100,Welding_Offset {X 0.0,Y 0.0,Z 0.0}}
L180_Welding_Craft[2,8]={Welding_Name[] "S8",Welding_Pos {X 533.000,Y 463.600037,Z -2.05000,A 0.0,B -23.0000,C 0.0},Welding_Power 80.0000,Welding_Speed 0.0400000,Welding_Angle -20.0000,Welding_CDIS 5,Welding_ACC 100,Welding_Offset {X 0.0,Y 0.0,Z 0.0}}
L180_Welding_Craft[2,9]={Welding_Name[] "S9",Welding_Pos {X 533.000,Y 463.600037,Z -2.05000,A 0.0,B -23.0000,C 0.0},Welding_Power 80.0000,Welding_Speed 0.0400000,Welding_Angle -20.0000,Welding_CDIS 5,Welding_ACC 100,Welding_Offset {X 0.0,Y 0.0,Z 0.0}}
L180_Welding_Craft[2,10]={Welding_Name[] "S10",Welding_Pos {X 533.000,Y 338.000,Z -2.05000,A 0.0,B -23.0000,C 0.0},Welding_Power 80.0000,Welding_Speed 0.0400000,Welding_Angle -20.0000,Welding_CDIS 5,Welding_ACC 100,Welding_Offset {X 0.0,Y 0.0,Z 0.0}}

DECL GLOBAL Surr_Welding_Craft_Type C225_Welding_Craft[2,3]
C225_Welding_Craft[1,1]={Welding_Name[] "S3",Welding_Pos {X 20.0000,Y 110.000,Z 0.0,A 0.0,B -20.0000,C 0.0},Welding_Power 80.0000,Welding_Speed 0.0400000,Welding_Angle -20.0000,Welding_CDIS 5,Welding_ACC 100,Welding_Offset {X 0.0,Y 0.0,Z 0.0}}
C225_Welding_Craft[1,2]={Welding_Name[] "PM3",Welding_Pos {X 22.9300,Y 117.070,Z 0.0,A 0.0,B 0.0,C 0.0},Welding_Power 80.0000,Welding_Speed 0.0400000,Welding_Angle -20.0000,Welding_CDIS 5,Welding_ACC 100,Welding_Offset {X 0.0,Y 0.0,Z 0.0},Welding_Offset_CIR {C_X 0.0,C_Y 0.0,C_Z 0.0}}
C225_Welding_Craft[1,3]={Welding_Name[] "PE3",Welding_Pos {X 30.0000,Y 120.000,Z 0.0,A 0.0,B 0.0,C -20.0000},Welding_Power 80.0000,Welding_Speed 0.0400000,Welding_Angle -20.0000,Welding_CDIS 5,Welding_ACC 100,Welding_Offset {X 0.0,Y 0.0,Z 0.0}}
C225_Welding_Craft[2,1]={Welding_Name[] "C225_S1",Welding_Pos {X 23.2174511,Y 715.439,Z 0.0,A 0.0,B -20.0000,C 0.0},Welding_Power 80.0000,Welding_Speed 0.0300000,Welding_Angle -20.0000,Welding_CDIS 5,Welding_ACC 100,Welding_Offset {X 0.300000,Y 0.0,Z 0.0}}
C225_Welding_Craft[2,2]={Welding_Name[] "PM5",Welding_Pos {X 27.1170,Y 722.236,Z 0.0,A 0.0,B 0.0,C 0.0},Welding_Power 80.0000,Welding_Speed 0.0400000,Welding_Angle -20.0000,Welding_CDIS 5,Welding_ACC 100,Welding_Offset {X 0.0,Y 0.0,Z 0.0},Welding_Offset_CIR {C_X 0.0,C_Y 0.0,C_Z 0.0}}
C225_Welding_Craft[2,3]={Welding_Name[] "PE5",Welding_Pos {X 33.2110,Y 725.443054,Z 0.0,A 0.0,B 0.0,C -20.0000},Welding_Power 80.0000,Welding_Speed 0.0150000,Welding_Angle -20.0000,Welding_CDIS 5,Welding_ACC 100,Welding_Offset {X 0.0,Y 0.0,Z 0.0}}

DECL GLOBAL Surr_Welding_Craft_Type L270_Welding_Craft[2,10]
L270_Welding_Craft[1,1]={Welding_Name[] "S2",Welding_Pos {X 110.000,Y 120.000,Z 0.0,A 0.0,B 0.0,C -20.0000},Welding_Power 80.0000,Welding_Speed 0.0400000,Welding_Angle -20.0000,Welding_CDIS 5,Welding_ACC 100,Welding_Offset {X 0.0,Y 0.0,Z 0.0}}
L270_Welding_Craft[1,2]={Welding_Name[] "L270_S2",Welding_Pos {X 200.000,Y 656.000,Z 0.0,A 0.0,B 0.0,C -20.0000},Welding_Power 80.0000,Welding_Speed 0.0400000,Welding_Angle -20.0000,Welding_CDIS 5,Welding_ACC 100,Welding_Offset {X 0.0,Y 0.0,Z 0.0}}
L270_Welding_Craft[1,3]={Welding_Name[] "L270_S3",Welding_Pos {X 349.400,Y 656.000,Z 0.0,A 0.0,B 0.0,C -20.0000},Welding_Power 80.0000,Welding_Speed 0.0400000,Welding_Angle -20.0000,Welding_CDIS 5,Welding_ACC 100,Welding_Offset {X 0.0,Y 0.0,Z 0.0}}
L270_Welding_Craft[1,4]={Welding_Name[] "S4",Welding_Pos {X 400.000,Y 86.0000153,Z -3.00000,A 0.0,B 23.0000,C 0.0},Welding_Power 80.0000,Welding_Speed 0.0400000,Welding_Angle -20.0000,Welding_CDIS 5,Welding_ACC 100,Welding_Offset {X 0.0,Y 0.0,Z 0.0}}
L270_Welding_Craft[1,5]={Welding_Name[] "S12",Welding_Pos {X 28.9999981,Y 400.000,Z -3.00000,A 0.0,B 0.0,C -23.0000},Welding_Power 80.0000,Welding_Speed 0.0400000,Welding_Angle -20.0000,Welding_CDIS 5,Welding_ACC 100,Welding_Offset {X 0.0,Y 0.0,Z 0.0}}
L270_Welding_Craft[1,6]={Welding_Name[] "S6",Welding_Pos {X 533.000,Y 463.600037,Z -2.05000,A 0.0,B -23.0000,C 0.0},Welding_Power 80.0000,Welding_Speed 0.0400000,Welding_Angle -20.0000,Welding_CDIS 5,Welding_ACC 100,Welding_Offset {X 0.0,Y 0.0,Z 0.0}}
L270_Welding_Craft[1,7]={Welding_Name[] "S7",Welding_Pos {X 533.000,Y 463.600037,Z -2.05000,A 0.0,B -23.0000,C 0.0},Welding_Power 80.0000,Welding_Speed 0.0400000,Welding_Angle -20.0000,Welding_CDIS 5,Welding_ACC 100,Welding_Offset {X 0.0,Y 0.0,Z 0.0}}
L270_Welding_Craft[1,8]={Welding_Name[] "S8",Welding_Pos {X 533.000,Y 463.600037,Z -2.05000,A 0.0,B -23.0000,C 0.0},Welding_Power 80.0000,Welding_Speed 0.0400000,Welding_Angle -20.0000,Welding_CDIS 5,Welding_ACC 100,Welding_Offset {X 0.0,Y 0.0,Z 0.0}}
L270_Welding_Craft[1,9]={Welding_Name[] "S9",Welding_Pos {X 533.000,Y 463.600037,Z -2.05000,A 0.0,B -23.0000,C 0.0},Welding_Power 80.0000,Welding_Speed 0.0400000,Welding_Angle -20.0000,Welding_CDIS 5,Welding_ACC 100,Welding_Offset {X 0.0,Y 0.0,Z 0.0}}
L270_Welding_Craft[1,10]={Welding_Name[] "S10",Welding_Pos {X 533.000,Y 338.000,Z -2.05000,A 0.0,B -23.0000,C 0.0},Welding_Power 80.0000,Welding_Speed 0.0400000,Welding_Angle -20.0000,Welding_CDIS 5,Welding_ACC 100,Welding_Offset {X 0.0,Y 0.0,Z 0.0}}
L270_Welding_Craft[2,1]={Welding_Name[] "L270_S1",Welding_Pos {X 66.4440918,Y 725.456543,Z 0.0,A 0.0,B 0.0,C -20.0000},Welding_Power 80.0000,Welding_Speed 0.0320000,Welding_Angle -20.0000,Welding_CDIS 5,Welding_ACC 100,Welding_Offset {X 0.0,Y 0.0,Z 0.0}}
L270_Welding_Craft[2,2]={Welding_Name[] "L270_S2",Welding_Pos {X 199.376495,Y 725.510498,Z 0.0,A 0.0,B 0.0,C -20.0000},Welding_Power 80.0000,Welding_Speed 0.0320000,Welding_Angle -20.0000,Welding_CDIS 5,Welding_ACC 100,Welding_Offset {X 0.0,Y 0.0,Z 0.0}}
L270_Welding_Craft[2,3]={Welding_Name[] "L270_S3",Welding_Pos {X 348.925446,Y 725.571167,Z 0.0,A 0.0,B 0.0,C -20.0000},Welding_Power 80.0000,Welding_Speed 0.0320000,Welding_Angle -20.0000,Welding_CDIS 5,Welding_ACC 100,Welding_Offset {X 0.0,Y 0.0,Z 0.0}}
L270_Welding_Craft[2,4]={Welding_Name[] "S4",Welding_Pos {X 400.000,Y 86.0000153,Z -3.00000,A 0.0,B 23.0000,C 0.0},Welding_Power 80.0000,Welding_Speed 0.0400000,Welding_Angle -20.0000,Welding_CDIS 5,Welding_ACC 100,Welding_Offset {X 0.0,Y 0.0,Z 0.0}}
L270_Welding_Craft[2,5]={Welding_Name[] "S12",Welding_Pos {X 28.9999981,Y 400.000,Z -3.00000,A 0.0,B 0.0,C -23.0000},Welding_Power 80.0000,Welding_Speed 0.0400000,Welding_Angle -20.0000,Welding_CDIS 5,Welding_ACC 100,Welding_Offset {X 0.0,Y 0.0,Z 0.0}}
L270_Welding_Craft[2,6]={Welding_Name[] "S6",Welding_Pos {X 533.000,Y 463.600037,Z -2.05000,A 0.0,B -23.0000,C 0.0},Welding_Power 80.0000,Welding_Speed 0.0400000,Welding_Angle -20.0000,Welding_CDIS 5,Welding_ACC 100,Welding_Offset {X 0.0,Y 0.0,Z 0.0}}
L270_Welding_Craft[2,7]={Welding_Name[] "S7",Welding_Pos {X 533.000,Y 463.600037,Z -2.05000,A 0.0,B -23.0000,C 0.0},Welding_Power 80.0000,Welding_Speed 0.0400000,Welding_Angle -20.0000,Welding_CDIS 5,Welding_ACC 100,Welding_Offset {X 0.0,Y 0.0,Z 0.0}}
L270_Welding_Craft[2,8]={Welding_Name[] "S8",Welding_Pos {X 533.000,Y 463.600037,Z -2.05000,A 0.0,B -23.0000,C 0.0},Welding_Power 80.0000,Welding_Speed 0.0400000,Welding_Angle -20.0000,Welding_CDIS 5,Welding_ACC 100,Welding_Offset {X 0.0,Y 0.0,Z 0.0}}
L270_Welding_Craft[2,9]={Welding_Name[] "S9",Welding_Pos {X 533.000,Y 463.600037,Z -2.05000,A 0.0,B -23.0000,C 0.0},Welding_Power 80.0000,Welding_Speed 0.0400000,Welding_Angle -20.0000,Welding_CDIS 5,Welding_ACC 100,Welding_Offset {X 0.0,Y 0.0,Z 0.0}}
L270_Welding_Craft[2,10]={Welding_Name[] "S10",Welding_Pos {X 533.000,Y 338.000,Z -2.05000,A 0.0,B -23.0000,C 0.0},Welding_Power 80.0000,Welding_Speed 0.0400000,Welding_Angle -20.0000,Welding_CDIS 5,Welding_ACC 100,Welding_Offset {X 0.0,Y 0.0,Z 0.0}}

DECL GLOBAL Surr_Welding_Craft_Type C315_Welding_Craft[2,3]
C315_Welding_Craft[1,1]={Welding_Name[] "C315_S1",Welding_Pos {X 366.000,Y 656.000,Z 0.0,A 0.0,B 0.0,C -20.0000},Welding_Power 80.0000,Welding_Speed 0.0400000,Welding_Angle -20.0000,Welding_CDIS 5,Welding_ACC 100,Welding_Offset {X 0.0,Y 0.0,Z 0.0}}
C315_Welding_Craft[1,2]={Welding_Name[] "PM3",Welding_Pos {X 373.071075,Y 653.071045,Z 0.0,A 0.0,B 0.0,C 0.0},Welding_Power 80.0000,Welding_Speed 0.0400000,Welding_Angle 20.0000,Welding_CDIS 5,Welding_ACC 100,Welding_Offset {X 0.0,Y 0.0,Z 0.0},Welding_Offset_CIR {C_X 0.0,C_Y 0.0,C_Z 0.0}}
C315_Welding_Craft[1,3]={Welding_Name[] "PE5",Welding_Pos {X 376.000,Y 646.000,Z 0.0,A 0.0,B 20.0000,C 0.0},Welding_Power 80.0000,Welding_Speed 0.0400000,Welding_Angle 20.0000,Welding_CDIS 5,Welding_ACC 100,Welding_Offset {X 0.0,Y 0.0,Z 0.0}}
C315_Welding_Craft[2,1]={Welding_Name[] "C315_S1",Welding_Pos {X 365.542,Y 725.577942,Z 0.0,A 0.0,B 0.0,C -20.0000},Welding_Power 80.0000,Welding_Speed 0.0300000,Welding_Angle -20.0000,Welding_CDIS 5,Welding_ACC 100,Welding_Offset {X 0.0,Y 0.0,Z 0.0}}
C315_Welding_Craft[2,2]={Welding_Name[] "PM7",Welding_Pos {X 371.833,Y 722.250,Z 0.0,A 0.0,B 0.0,C 0.0},Welding_Power 80.0000,Welding_Speed 0.0400000,Welding_Angle 20.0000,Welding_CDIS 5,Welding_ACC 100,Welding_Offset {X 0.0,Y 0.0,Z 0.0},Welding_Offset_CIR {C_X 0.0,C_Y 0.0,C_Z 0.0}}
C315_Welding_Craft[2,3]={Welding_Name[] "PE7",Welding_Pos {X 375.545074,Y 715.582,Z 0.0,A 0.0,B 20.0000,C 0.0},Welding_Power 80.0000,Welding_Speed 0.0150000,Welding_Angle 20.0000,Welding_CDIS 5,Welding_ACC 100,Welding_Offset {X -1.00000,Y 0.0,Z 0.0}}


DECL GLOBAL Surr_Welding_Craft_Type N45_Short_Craft[2,5]
N45_Short_Craft[1,1]={Welding_Name[] "S2",Welding_Pos {X 364.000,Y 0.0,Z -150.000,A 0.0,B 0.0,C 0.0},Welding_Power 80.0000,Welding_Speed 0.500000,Welding_Angle 0.0,Welding_CDIS 0,Welding_ACC 100,Welding_Offset {X 0.0,Y 0.0,Z 0.0}}
N45_Short_Craft[1,2]={Welding_Name[] "S13",Welding_Pos {X 364.000,Y 0.0,Z 0.0,A 0.0,B 0.0,C 0.0},Welding_Power 80.0000,Welding_Speed 0.500000,Welding_Angle 0.0,Welding_CDIS 0,Welding_ACC 100,Welding_Offset {X 0.0,Y 0.0,Z 0.0}}
N45_Short_Craft[1,3]={Welding_Name[] "S14",Welding_Pos {X 364.000,Y 23.0000,Z 0.0,A 0.0,B 0.0,C 0.0},Welding_Power 80.0000,Welding_Speed 0.01000000,Welding_Angle 0.0,Welding_CDIS 0,Welding_ACC 100,Welding_Offset {X 0.0,Y 0.0,Z 0.0}}
N45_Short_Craft[1,4]={Welding_Name[] "S4",Welding_Pos {X 364.000,Y 20.7000,Z -150.000,A 0.0,B 0.0,C 0.0},Welding_Power 80.0000,Welding_Speed 0.500000,Welding_Angle 0.0,Welding_CDIS 0,Welding_ACC 100,Welding_Offset {X 0.0,Y 0.0,Z 0.0}}
N45_Short_Craft[1,5]={Welding_Name[] "S12",Welding_Pos {X 28.9999981,Y 400.000,Z -3.00000,A 0.0,B 0.0,C -23.0000},Welding_Power 80.0000,Welding_Speed 0.500000,Welding_Angle 0.0,Welding_CDIS 0,Welding_ACC 100,Welding_Offset {X 0.0,Y 0.0,Z 0.0}}
N45_Short_Craft[2,1]={Welding_Name[] "S32",Welding_Pos {X 363.220,Y -0.316000,Z -150.000,A 0.0,B 0.0,C 0.0},Welding_Power 80.0000,Welding_Speed 0.500000,Welding_Angle 0.0,Welding_CDIS 0,Welding_ACC 100,Welding_Offset {X 0.0,Y 0.0,Z 0.0}}
N45_Short_Craft[2,2]={Welding_Name[] "S13",Welding_Pos {X 363.220,Y -0.316000,Z 0.0,A 0.0,B 0.0,C 0.0},Welding_Power 80.0000,Welding_Speed 0.500000,Welding_Angle 0.0,Welding_CDIS 0,Welding_ACC 100,Welding_Offset {X 0.0,Y 0.0,Z 0.0}}
N45_Short_Craft[2,3]={Welding_Name[] "S14",Welding_Pos {X 363.395,Y 19.3140,Z 0.0,A 0.0,B 0.0,C 0.0},Welding_Power 80.0000,Welding_Speed 0.01000000,Welding_Angle 0.0,Welding_CDIS 0,Welding_ACC 100,Welding_Offset {X 0.0,Y 0.0,Z 0.0}}
N45_Short_Craft[2,4]={Welding_Name[] "S4",Welding_Pos {X 363.323059,Y 11.2466183,Z -150.000,A 0.0,B 0.0,C 0.0},Welding_Power 80.0000,Welding_Speed 0.500000,Welding_Angle 0.0,Welding_CDIS 0,Welding_ACC 100,Welding_Offset {X 0.0,Y 0.0,Z 0.0}}
N45_Short_Craft[2,5]={Welding_Name[] "S12",Welding_Pos {X 28.9999981,Y 400.000,Z -3.00000,A 0.0,B 0.0,C -23.0000},Welding_Power 80.0000,Welding_Speed 0.500000,Welding_Angle 0.0,Welding_CDIS 0,Welding_ACC 100,Welding_Offset {X 0.0,Y 0.0,Z 0.0}}

DECL GLOBAL Surr_Welding_Craft_Type N135_Short_Craft[2,5]
N135_Short_Craft[1,1]={Welding_Name[] "S9",Welding_Pos {X 36.0000,Y 0.0,Z -150.000,A 0.0,B 0.0,C 0.0},Welding_Power 80.0000,Welding_Speed 0.500000,Welding_Angle 0.0,Welding_CDIS 0,Welding_ACC 100,Welding_Offset {X 0.0,Y 0.0,Z 0.0}}
N135_Short_Craft[1,2]={Welding_Name[] "S13",Welding_Pos {X 36.0000,Y 0.0,Z 0.0,A 0.0,B 0.0,C 0.0},Welding_Power 80.0000,Welding_Speed 0.500000,Welding_Angle 0.0,Welding_CDIS 0,Welding_ACC 100,Welding_Offset {X 0.0,Y 0.0,Z 0.0}}
N135_Short_Craft[1,3]={Welding_Name[] "S14",Welding_Pos {X 36.0000,Y 23.0000,Z 0.0,A 0.0,B 0.0,C 0.0},Welding_Power 80.0000,Welding_Speed 0.01000000,Welding_Angle 0.0,Welding_CDIS 0,Welding_ACC 100,Welding_Offset {X 0.0,Y 0.0,Z 0.0}}
N135_Short_Craft[1,4]={Welding_Name[] "S4",Welding_Pos {X 36.0000,Y 20.7000,Z -150.000,A 0.0,B 0.0,C 0.0},Welding_Power 80.0000,Welding_Speed 0.500000,Welding_Angle 0.0,Welding_CDIS 0,Welding_ACC 100,Welding_Offset {X 0.0,Y 0.0,Z 0.0}}
N135_Short_Craft[1,5]={Welding_Name[] "S12",Welding_Pos {X 28.9999981,Y 400.000,Z -3.00000,A 0.0,B 0.0,C -23.0000},Welding_Power 80.0000,Welding_Speed 0.500000,Welding_Angle 0.0,Welding_CDIS 0,Welding_ACC 100,Welding_Offset {X 0.0,Y 0.0,Z 0.0}}
N135_Short_Craft[2,1]={Welding_Name[] "S92",Welding_Pos {X 32.5260,Y -0.971000,Z -150.000,A 0.0,B 0.0,C 0.0},Welding_Power 80.0000,Welding_Speed 0.500000,Welding_Angle 0.0,Welding_CDIS 0,Welding_ACC 100,Welding_Offset {X 0.0,Y 0.0,Z 0.0}}
N135_Short_Craft[2,2]={Welding_Name[] "S13",Welding_Pos {X 32.5260,Y -0.971000,Z 0.0,A 0.0,B 0.0,C 0.0},Welding_Power 80.0000,Welding_Speed 0.500000,Welding_Angle 0.0,Welding_CDIS 0,Welding_ACC 100,Welding_Offset {X 0.0,Y 0.0,Z 0.0}}
N135_Short_Craft[2,3]={Welding_Name[] "S14",Welding_Pos {X 32.3940,Y 18.1940,Z 0.0,A 0.0,B 0.0,C 0.0},Welding_Power 80.0000,Welding_Speed 0.01000000,Welding_Angle 0.0,Welding_CDIS 0,Welding_ACC 100,Welding_Offset {X 0.0,Y 0.0,Z 0.0}}
N135_Short_Craft[2,4]={Welding_Name[] "S4",Welding_Pos {X 32.4600,Y 8.61150074,Z -150.000,A 0.0,B 0.0,C 0.0},Welding_Power 80.0000,Welding_Speed 0.500000,Welding_Angle 0.0,Welding_CDIS 0,Welding_ACC 100,Welding_Offset {X 0.0,Y 0.0,Z 0.0}}
N135_Short_Craft[2,5]={Welding_Name[] "S12",Welding_Pos {X 28.9999981,Y 400.000,Z -3.00000,A 0.0,B 0.0,C -23.0000},Welding_Power 80.0000,Welding_Speed 0.500000,Welding_Angle 0.0,Welding_CDIS 0,Welding_ACC 100,Welding_Offset {X 0.0,Y 0.0,Z 0.0}}

DECL GLOBAL Surr_Welding_Craft_Type N225_Short_Craft[2,5]
N225_Short_Craft[1,1]={Welding_Name[] "S10",Welding_Pos {X 36.0000,Y 680.000,Z -150.000,A 0.0,B 0.0,C 0.0},Welding_Power 80.0000,Welding_Speed 0.500000,Welding_Angle 0.0,Welding_CDIS 0,Welding_ACC 100,Welding_Offset {X 0.0,Y 0.0,Z 0.0}}
N225_Short_Craft[1,2]={Welding_Name[] "S13",Welding_Pos {X 36.0000,Y 680.000,Z 0.0,A 0.0,B 0.0,C 0.0},Welding_Power 80.0000,Welding_Speed 0.500000,Welding_Angle 0.0,Welding_CDIS 0,Welding_ACC 100,Welding_Offset {X 0.0,Y 0.0,Z 0.0}}
N225_Short_Craft[1,3]={Welding_Name[] "S14",Welding_Pos {X 36.0000,Y 657.000,Z 0.0,A 0.0,B 0.0,C 0.0},Welding_Power 80.0000,Welding_Speed 0.01000000,Welding_Angle 0.0,Welding_CDIS 0,Welding_ACC 100,Welding_Offset {X 0.0,Y 0.0,Z 0.0}}
N225_Short_Craft[1,4]={Welding_Name[] "S4",Welding_Pos {X 36.0000,Y 667.500,Z -150.000,A 0.0,B 0.0,C 0.0},Welding_Power 80.0000,Welding_Speed 0.500000,Welding_Angle 0.0,Welding_CDIS 0,Welding_ACC 100,Welding_Offset {X 0.0,Y 0.0,Z 0.0}}
N225_Short_Craft[1,5]={Welding_Name[] "S12",Welding_Pos {X 28.9999981,Y 400.000,Z -3.00000,A 0.0,B 0.0,C -23.0000},Welding_Power 80.0000,Welding_Speed 0.500000,Welding_Angle 0.0,Welding_CDIS 0,Welding_ACC 100,Welding_Offset {X 0.0,Y 0.0,Z 0.0}}
N225_Short_Craft[2,1]={Welding_Name[] "S13",Welding_Pos {X 31.6330,Y 679.439,Z -150.000,A 0.0,B 0.0,C 0.0},Welding_Power 80.0000,Welding_Speed 0.500000,Welding_Angle 0.0,Welding_CDIS 0,Welding_ACC 100,Welding_Offset {X 0.0,Y 0.0,Z 0.0}}
N225_Short_Craft[2,2]={Welding_Name[] "S13",Welding_Pos {X 31.6330,Y 679.439,Z 0.0,A 0.0,B 0.0,C 0.0},Welding_Power 80.0000,Welding_Speed 0.500000,Welding_Angle 0.0,Welding_CDIS 0,Welding_ACC 100,Welding_Offset {X 0.0,Y 0.0,Z 0.0}}
N225_Short_Craft[2,3]={Welding_Name[] "S14",Welding_Pos {X 31.8670,Y 660.025,Z 0.0,A 0.0,B 0.0,C 0.0},Welding_Power 80.0000,Welding_Speed 0.01000000,Welding_Angle 0.0,Welding_CDIS 0,Welding_ACC 100,Welding_Offset {X 0.0,Y 0.0,Z 0.0}}
N225_Short_Craft[2,4]={Welding_Name[] "S4",Welding_Pos {X 31.7500,Y 669.732056,Z -150.000,A 0.0,B 0.0,C 0.0},Welding_Power 80.0000,Welding_Speed 0.500000,Welding_Angle 0.0,Welding_CDIS 0,Welding_ACC 100,Welding_Offset {X 0.0,Y 0.0,Z 0.0}}
N225_Short_Craft[2,5]={Welding_Name[] "S12",Welding_Pos {X 28.9999981,Y 400.000,Z -3.00000,A 0.0,B 0.0,C -23.0000},Welding_Power 80.0000,Welding_Speed 0.500000,Welding_Angle 0.0,Welding_CDIS 0,Welding_ACC 100,Welding_Offset {X 0.0,Y 0.0,Z 0.0}}

DECL GLOBAL Surr_Welding_Craft_Type N315_Short_Craft[2,5]
N315_Short_Craft[1,1]={Welding_Name[] "S17",Welding_Pos {X 364.000,Y 680.000,Z -150.000,A 0.0,B 0.0,C 0.0},Welding_Power 80.0000,Welding_Speed 0.500000,Welding_Angle 0.0,Welding_CDIS 0,Welding_ACC 100,Welding_Offset {X 0.0,Y 0.0,Z 0.0}}
N315_Short_Craft[1,2]={Welding_Name[] "S13",Welding_Pos {X 364.000,Y 680.000,Z 0.0,A 0.0,B 0.0,C 0.0},Welding_Power 80.0000,Welding_Speed 0.500000,Welding_Angle 0.0,Welding_CDIS 0,Welding_ACC 100,Welding_Offset {X 0.0,Y 0.0,Z 0.0}}
N315_Short_Craft[1,3]={Welding_Name[] "S14",Welding_Pos {X 364.000,Y 657.000,Z 0.0,A 0.0,B 0.0,C 0.0},Welding_Power 80.0000,Welding_Speed 0.01000000,Welding_Angle 0.0,Welding_CDIS 0,Welding_ACC 100,Welding_Offset {X 0.0,Y 0.0,Z 0.0}}
N315_Short_Craft[1,4]={Welding_Name[] "S4",Welding_Pos {X 364.000,Y 667.500,Z -150.000,A 0.0,B 0.0,C 0.0},Welding_Power 80.0000,Welding_Speed 0.500000,Welding_Angle 0.0,Welding_CDIS 0,Welding_ACC 100,Welding_Offset {X 0.0,Y 0.0,Z 0.0}}
N315_Short_Craft[1,5]={Welding_Name[] "S12",Welding_Pos {X 28.9999981,Y 400.000,Z -3.00000,A 0.0,B 0.0,C -23.0000},Welding_Power 80.0000,Welding_Speed 0.500000,Welding_Angle 0.0,Welding_CDIS 0,Welding_ACC 100,Welding_Offset {X 0.0,Y 0.0,Z 0.0}}
N315_Short_Craft[2,1]={Welding_Name[] "S17",Welding_Pos {X 362.986,Y 679.910,Z -150.000,A 0.0,B 0.0,C 0.0},Welding_Power 80.0000,Welding_Speed 0.500000,Welding_Angle 0.0,Welding_CDIS 0,Welding_ACC 100,Welding_Offset {X 0.0,Y 0.0,Z 0.0}}
N315_Short_Craft[2,2]={Welding_Name[] "S13",Welding_Pos {X 362.986,Y 679.910,Z 0.0,A 0.0,B 0.0,C 0.0},Welding_Power 80.0000,Welding_Speed 0.500000,Welding_Angle 0.0,Welding_CDIS 0,Welding_ACC 100,Welding_Offset {X 0.0,Y 0.0,Z 0.0}}
N315_Short_Craft[2,3]={Welding_Name[] "S14",Welding_Pos {X 363.044,Y 660.468,Z 0.0,A 0.0,B 0.0,C 0.0},Welding_Power 80.0000,Welding_Speed 0.01000000,Welding_Angle 0.0,Welding_CDIS 0,Welding_ACC 100,Welding_Offset {X 0.0,Y 0.0,Z 0.0}}
N315_Short_Craft[2,4]={Welding_Name[] "S4",Welding_Pos {X 363.015,Y 670.188965,Z -150.000,A 0.0,B 0.0,C 0.0},Welding_Power 80.0000,Welding_Speed 0.500000,Welding_Angle 0.0,Welding_CDIS 0,Welding_ACC 100,Welding_Offset {X 0.0,Y 0.0,Z 0.0}}
N315_Short_Craft[2,5]={Welding_Name[] "S12",Welding_Pos {X 28.9999981,Y 400.000,Z -3.00000,A 0.0,B 0.0,C -23.0000},Welding_Power 80.0000,Welding_Speed 0.500000,Welding_Angle 0.0,Welding_CDIS 0,Welding_ACC 100,Welding_Offset {X 0.0,Y 0.0,Z 0.0}}



DECL GLOBAL Surround_Welding_Type N1_Sink_Data={Sink_Size_Long 632.000,Sink_Size_Width 347.000,Sink_Size_R 12.0000,Sink_Size_Short_Side 23.0000,Sink_Size_Short_OnePos 36.0000,Sink_Size_Short_TwoPos 323.000,Sink_Size_Pots_Thick 0.0,Sink_Size_Panel_Thick 0.0,Sink_Model 952128,Sink_Size_Left_Distance 24.0000,Sink_Size_Down_Distance 24.0000,Sink_Type #LeftRight_One}
DECL GLOBAL Surround_Welding_Type N2_Sink_Data={Sink_Size_Long 700.000,Sink_Size_Width 350.000,Sink_Size_R 10.0000,Sink_Size_Short_Side 23.0000,Sink_Size_Short_OnePos 36.0000,Sink_Size_Short_TwoPos 328.000,Sink_Size_Pots_Thick 0.0,Sink_Size_Panel_Thick 0.0,Sink_Model 952212,Sink_Size_Left_Distance 25.0000,Sink_Size_Down_Distance 25.0000,Sink_Type #LeftRight_One}
;-----------Viion_INI------------



DECL GLOBAL INT Vision_Scope=20
;GLOBAL CHAR $Socket_Connect[1024]
;DECL GLOBAL CHAR $SOCKET_MESS[1024]
;DECL GLOBAL MODEL_TYPE $N_1
;DECL GLOBAL MODEL_TYPE $N_2
;DECL GLOBAL INT $MY_Work_Number=-1



;----------------------------------
ENDDAT
